REGION Network 98: MENSAJES - AUSENCIA
   RUNG wire#powerrail
      Contact( #Mx_ET151 )
      Contact( #Mx_ET51 )
      wire#w1
      I_Contact( #pHsMx_1 )
      I_Contact( #pHsMx_2 )
      I_Contact( #pHsMx_3 )
      I_Contact( #pHsMx_4 )
      S_SR(operand := #STAT_EnvMens_AMx, r1 := wire#w2)
      Coil( #P_EnvMens_AMx )
   END_RUNG
   RUNG wire#powerrail
      Contact( #Mx_ET161 )
      Contact( #Mx_ET61 )
   END_RUNG wire#w1
   RUNG wire#powerrail
      I_Contact( #Mx_ET151 )
      I_Contact( #Mx_ET161 )
   END_RUNG wire#w2
   // the same network as SCL:
   IF ((#Mx_ET151 AND #Mx_ET51) OR (#Mx_ET161 AND #Mx_ET61)) AND NOT #pHsMx_1 AND NOT #pHsMx_2 AND NOT #pHsMx_3 AND NOT #pHsMx_4 THEN
       #STAT_EnvMens_AMx := TRUE;   // SR flip-flop
   END_IF;
   IF NOT #Mx_ET151 AND NOT #Mx_ET161 THEN #STAT_EnvMens_AMx := FALSE; END_IF;
   #P_EnvMens_AMx := #STAT_EnvMens_AMx;
END_REGION

REGION Network 99: MENSAJES - RECIBIDA LA ORDEN
   RUNG wire#powerrail
      Contact( #Mx_ET150 )
      I_Contact( #Mx_ET50 )
      wire#w1
      Coil( #P_RecepOK_Mx )
   END_RUNG
   RUNG wire#powerrail
      Contact( #Mx_ET160 )
      I_Contact( #Mx_ET60 )
   END_RUNG wire#w1
   // the same network as SCL:
   #P_RecepOK_Mx := (#Mx_ET150 AND NOT #Mx_ET50) OR (#Mx_ET160 AND NOT #Mx_ET60);
END_REGION

REGION Network 100: SALIDAS - Interlock FSS >> PickUp por S1
   RUNG wire#powerrail
      Contact( #Mx_ET60 )
      wire#w1
      Contact( #Pos_TROK )
      Contact( #Pos_TPOK )
      I_Contact( #Activado_Pasarela )
      Contact( #EstadoZona.Marcha_CBx )
      I_Contact( #EstadoVI.Error_Mx )
      I_Contact( #Error_Tx )
      Coil( #MA_PickUpOK_S1 )
   END_RUNG
   RUNG wire#powerrail
      Contact( #Mx_ET61 )
   END_RUNG wire#w1
   RUNG wire#powerrail
      Contact( #Mx_ET261 )
      I_Contact( #EstadoZona.ParoBlando_CBx )
   END_RUNG wire#w1
   // the same network as SCL:
   #MA_PickUpOK_S1 := (#Mx_ET60 OR #Mx_ET61 OR (#Mx_ET261 AND NOT #EstadoZona.ParoBlando_CBx)) AND #Pos_TROK AND #Pos_TPOK AND NOT #Activado_Pasarela AND #EstadoZona.Marcha_CBx AND NOT #EstadoVI.Error_Mx AND NOT #Error_Tx;
END_REGION

REGION Network 101: SALIDAS - Interlock FSS >> PickUp por S3
   RUNG wire#powerrail
      Contact( #Mx_ET50 )
      wire#w1
      Contact( #Pos_TROK )
      Contact( #Pos_TPOK )
      I_Contact( #Activado_Pasarela )
      Contact( #EstadoZona.Marcha_CBx )
      I_Contact( #EstadoVI.Error_Mx )
      I_Contact( #Error_Tx )
      Coil( #MA_PickUpOK_S3 )
   END_RUNG
   RUNG wire#powerrail
      Contact( #Mx_ET51 )
   END_RUNG wire#w1
   RUNG wire#powerrail
      Contact( #Mx_ET261 )
      I_Contact( #EstadoZona.ParoBlando_CBx )
   END_RUNG wire#w1
   // the same network as SCL:
   #MA_PickUpOK_S3 := (#Mx_ET50 OR #Mx_ET51 OR (#Mx_ET261 AND NOT #EstadoZona.ParoBlando_CBx)) AND #Pos_TROK AND #Pos_TPOK AND NOT #Activado_Pasarela AND #EstadoZona.Marcha_CBx AND NOT #EstadoVI.Error_Mx AND NOT #Error_Tx;
END_REGION

REGION Network 102: VARIABLES INTERNAS - AVANCE DE CARGA
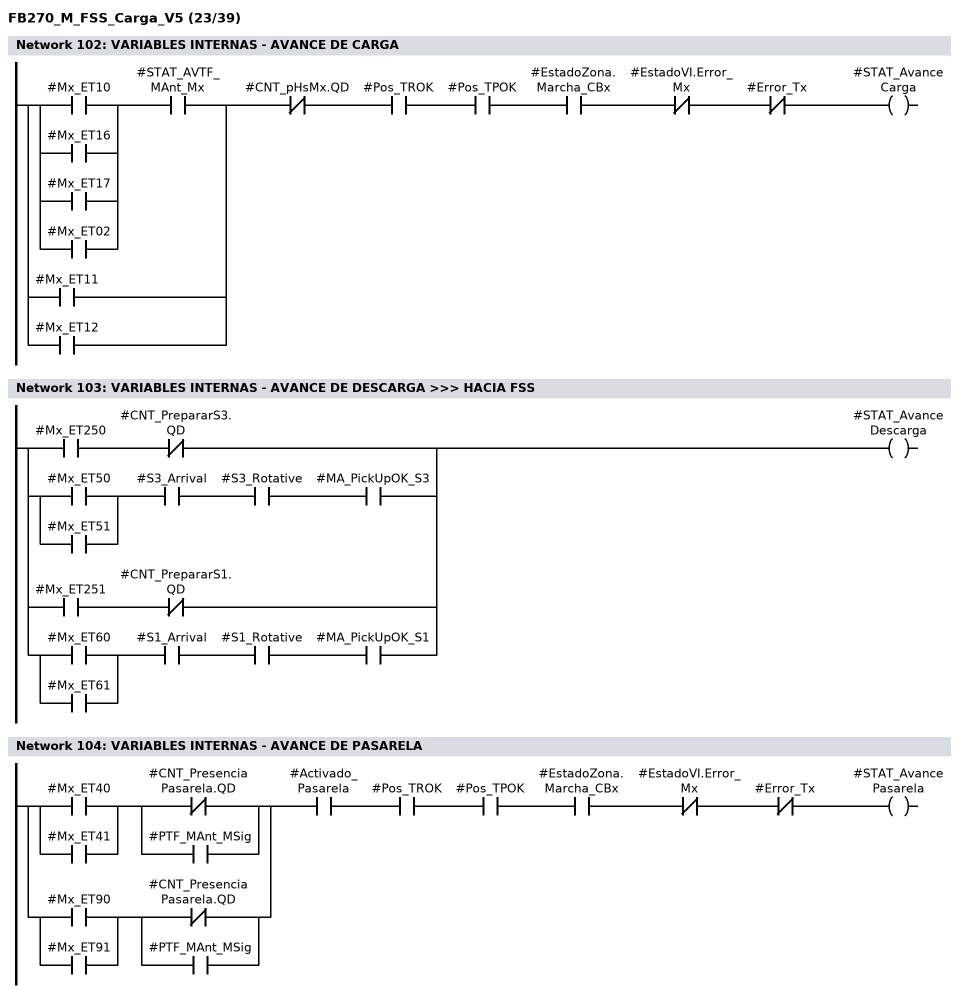
   RUNG wire#powerrail
      Contact( #Mx_ET10 )
      wire#w1
      Contact( #STAT_AVTF_MAnt_Mx )
      wire#w2
      I_Contact( #CNT_pHsMx.QD )
      Contact( #Pos_TROK )
      Contact( #Pos_TPOK )
      Contact( #EstadoZona.Marcha_CBx )
      I_Contact( #EstadoVI.Error_Mx )
      I_Contact( #Error_Tx )
      Coil( #STAT_AvanceCarga )
   END_RUNG
   RUNG wire#powerrail
      Contact( #Mx_ET16 )
   END_RUNG wire#w1
   RUNG wire#powerrail
      Contact( #Mx_ET17 )
   END_RUNG wire#w1
   RUNG wire#powerrail
      Contact( #Mx_ET02 )
   END_RUNG wire#w1
   RUNG wire#powerrail
      Contact( #Mx_ET11 )
   END_RUNG wire#w2
   RUNG wire#powerrail
      Contact( #Mx_ET12 )
   END_RUNG wire#w2
   // the same network as SCL:
   #STAT_AvanceCarga := (((#Mx_ET10 OR #Mx_ET16 OR #Mx_ET17 OR #Mx_ET02) AND #STAT_AVTF_MAnt_Mx) OR #Mx_ET11 OR #Mx_ET12) AND NOT #CNT_pHsMx.QD AND #Pos_TROK AND #Pos_TPOK AND #EstadoZona.Marcha_CBx AND NOT #EstadoVI.Error_Mx AND NOT #Error_Tx;
END_REGION

REGION Network 103: VARIABLES INTERNAS - AVANCE DE DESCARGA >>> HACIA FSS
   RUNG wire#powerrail
      Contact( #Mx_ET250 )
      I_Contact( #CNT_PrepararS3.QD )
      wire#w1
      Coil( #STAT_AvanceDescarga )
   END_RUNG
   RUNG wire#powerrail
      Contact( #Mx_ET50 )
      wire#w2
      Contact( #S3_Arrival )
      Contact( #S3_Rotative )
      Contact( #MA_PickUpOK_S3 )
   END_RUNG wire#w1
   RUNG wire#powerrail
      Contact( #Mx_ET51 )
   END_RUNG wire#w2
   RUNG wire#powerrail
      Contact( #Mx_ET251 )
      I_Contact( #CNT_PrepararS1.QD )
   END_RUNG wire#w1
   RUNG wire#powerrail
      Contact( #Mx_ET60 )
      wire#w3
      Contact( #S1_Arrival )
      Contact( #S1_Rotative )
      Contact( #MA_PickUpOK_S1 )
   END_RUNG wire#w1
   RUNG wire#powerrail
      Contact( #Mx_ET61 )
   END_RUNG wire#w3
   // the same network as SCL:
   #STAT_AvanceDescarga := (#Mx_ET250 AND NOT #CNT_PrepararS3.QD) OR ((#Mx_ET50 OR #Mx_ET51) AND #S3_Arrival AND #S3_Rotative AND #MA_PickUpOK_S3) OR (#Mx_ET251 AND NOT #CNT_PrepararS1.QD) OR ((#Mx_ET60 OR #Mx_ET61) AND #S1_Arrival AND #S1_Rotative AND #MA_PickUpOK_S1);
END_REGION

REGION Network 104: VARIABLES INTERNAS - AVANCE DE PASARELA
   RUNG wire#powerrail
      Contact( #Mx_ET40 )
      wire#w1
      I_Contact( #CNT_PresenciaPasarela.QD )
      wire#w2
      Contact( #Activado_Pasarela )
      Contact( #Pos_TROK )
      Contact( #Pos_TPOK )
      Contact( #EstadoZona.Marcha_CBx )
      I_Contact( #EstadoVI.Error_Mx )
      I_Contact( #Error_Tx )
      Coil( #STAT_AvancePasarela )
   END_RUNG
   RUNG wire#powerrail
      Contact( #Mx_ET41 )
   END_RUNG wire#w1
   RUNG wire#w1
      Contact( #PTF_MAnt_MSig )
   END_RUNG wire#w2
   RUNG wire#powerrail
      Contact( #Mx_ET90 )
      wire#w3
      I_Contact( #CNT_PresenciaPasarela.QD )
   END_RUNG wire#w2
   RUNG wire#powerrail
      Contact( #Mx_ET91 )
   END_RUNG wire#w3
   RUNG wire#w3
      Contact( #PTF_MAnt_MSig )
   END_RUNG wire#w2
   // the same network as SCL:
   #STAT_AvancePasarela := (((#Mx_ET40 OR #Mx_ET41) AND (NOT #CNT_PresenciaPasarela.QD OR #PTF_MAnt_MSig)) OR ((#Mx_ET90 OR #Mx_ET91) AND (NOT #CNT_PresenciaPasarela.QD OR #PTF_MAnt_MSig))) AND #Activado_Pasarela AND #Pos_TROK AND #Pos_TPOK AND #EstadoZona.Marcha_CBx AND NOT #EstadoVI.Error_Mx AND NOT #Error_Tx;
END_REGION

REGION Network 105: VARIABLES INTERNAS - VELOCIDAD BIT 00 >> RODILLOS 00-LenSima 01-Repos 10-Len 11-Rap
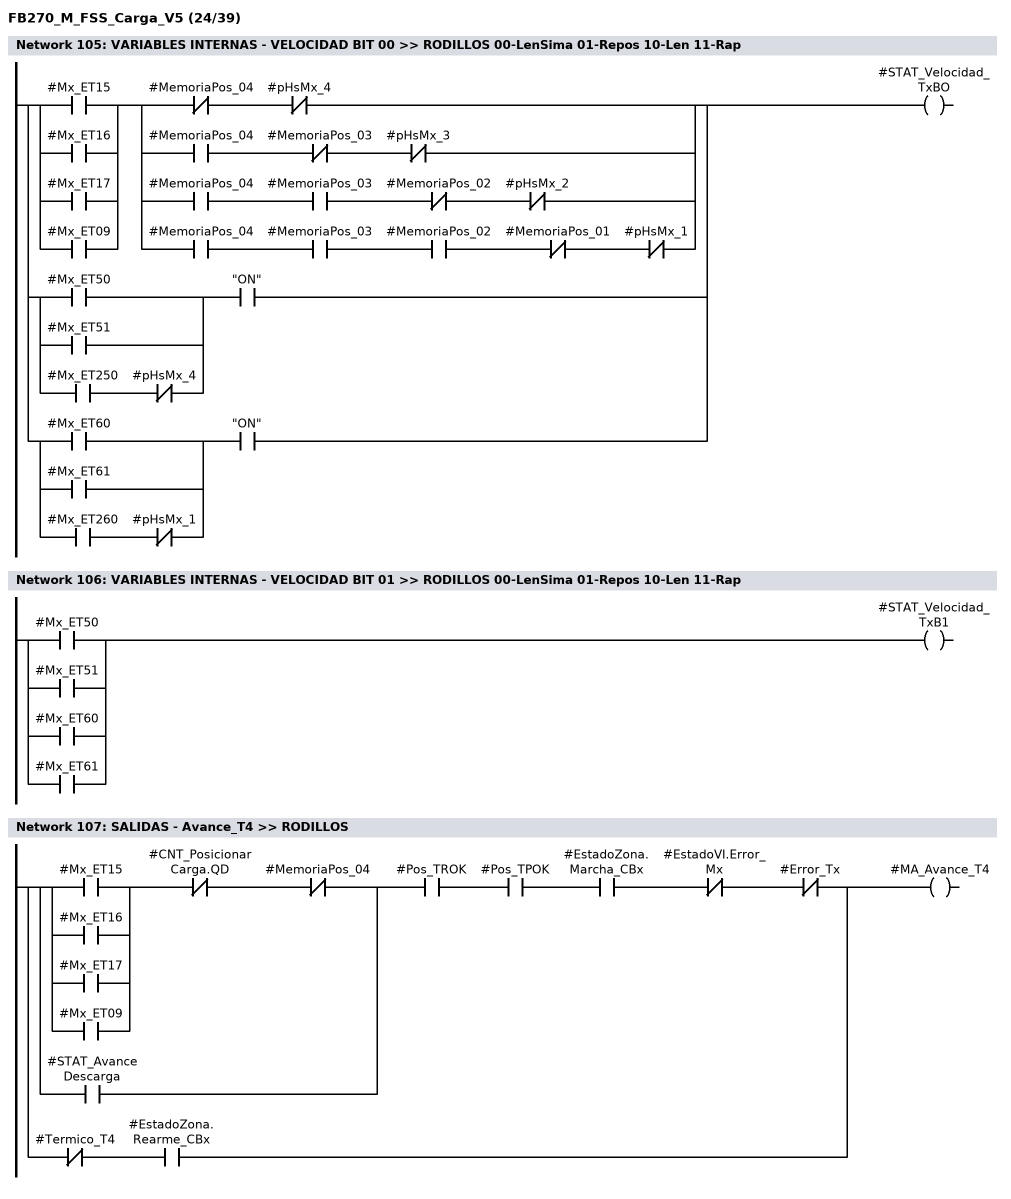
   RUNG wire#powerrail
      Contact( #Mx_ET15 )
      wire#w1
      I_Contact( #MemoriaPos_04 )
      I_Contact( #pHsMx_4 )
      wire#w2
      Coil( #STAT_Velocidad_TxBO )
   END_RUNG
   RUNG wire#powerrail
      Contact( #Mx_ET16 )
   END_RUNG wire#w1
   RUNG wire#powerrail
      Contact( #Mx_ET17 )
   END_RUNG wire#w1
   RUNG wire#powerrail
      Contact( #Mx_ET09 )
   END_RUNG wire#w1
   RUNG wire#w1
      Contact( #MemoriaPos_04 )
      I_Contact( #MemoriaPos_03 )
      I_Contact( #pHsMx_3 )
   END_RUNG wire#w2
   RUNG wire#w1
      Contact( #MemoriaPos_04 )
      Contact( #MemoriaPos_03 )
      I_Contact( #MemoriaPos_02 )
      I_Contact( #pHsMx_2 )
   END_RUNG wire#w2
   RUNG wire#w1
      Contact( #MemoriaPos_04 )
      Contact( #MemoriaPos_03 )
      Contact( #MemoriaPos_02 )
      I_Contact( #MemoriaPos_01 )
      I_Contact( #pHsMx_1 )
   END_RUNG wire#w2
   RUNG wire#powerrail
      Contact( #Mx_ET50 )
      wire#w3
      Contact( "ON" )
   END_RUNG wire#w2
   RUNG wire#powerrail
      Contact( #Mx_ET51 )
   END_RUNG wire#w3
   RUNG wire#powerrail
      Contact( #Mx_ET250 )
      I_Contact( #pHsMx_4 )
   END_RUNG wire#w3
   RUNG wire#powerrail
      Contact( #Mx_ET60 )
      wire#w4
      Contact( "ON" )
   END_RUNG wire#w2
   RUNG wire#powerrail
      Contact( #Mx_ET61 )
   END_RUNG wire#w4
   RUNG wire#powerrail
      Contact( #Mx_ET260 )
      I_Contact( #pHsMx_1 )
   END_RUNG wire#w4
   // the same network as SCL:
   #STAT_Velocidad_TxBO := ((#Mx_ET15 OR #Mx_ET16 OR #Mx_ET17 OR #Mx_ET09) AND ((NOT #MemoriaPos_04 AND NOT #pHsMx_4) OR (#MemoriaPos_04 AND NOT #MemoriaPos_03 AND NOT #pHsMx_3) OR (#MemoriaPos_04 AND #MemoriaPos_03 AND NOT #MemoriaPos_02 AND NOT #pHsMx_2) OR (#MemoriaPos_04 AND #MemoriaPos_03 AND #MemoriaPos_02 AND NOT #MemoriaPos_01 AND NOT #pHsMx_1))) OR ((#Mx_ET50 OR #Mx_ET51 OR (#Mx_ET250 AND NOT #pHsMx_4)) AND "ON") OR ((#Mx_ET60 OR #Mx_ET61 OR (#Mx_ET260 AND NOT #pHsMx_1)) AND "ON");
END_REGION

REGION Network 106: VARIABLES INTERNAS - VELOCIDAD BIT 01 >> RODILLOS 00-LenSima 01-Repos 10-Len 11-Rap
   RUNG wire#powerrail
      Contact( #Mx_ET50 )
      wire#w1
      Coil( #STAT_Velocidad_TxB1 )
   END_RUNG
   RUNG wire#powerrail
      Contact( #Mx_ET51 )
   END_RUNG wire#w1
   RUNG wire#powerrail
      Contact( #Mx_ET60 )
   END_RUNG wire#w1
   RUNG wire#powerrail
      Contact( #Mx_ET61 )
   END_RUNG wire#w1
   // the same network as SCL:
   #STAT_Velocidad_TxB1 := #Mx_ET50 OR #Mx_ET51 OR #Mx_ET60 OR #Mx_ET61;
END_REGION

REGION Network 107: SALIDAS - Avance_T4 >> RODILLOS
   RUNG wire#powerrail
      Contact( #Mx_ET15 )
      wire#w1
      I_Contact( #CNT_PosicionarCarga.QD )
      I_Contact( #MemoriaPos_04 )
      wire#w2
      Contact( #Pos_TROK )
      Contact( #Pos_TPOK )
      Contact( #EstadoZona.Marcha_CBx )
      I_Contact( #EstadoVI.Error_Mx )
      I_Contact( #Error_Tx )
      wire#w3
      Coil( #MA_Avance_T4 )
   END_RUNG
   RUNG wire#powerrail
      Contact( #Mx_ET16 )
   END_RUNG wire#w1
   RUNG wire#powerrail
      Contact( #Mx_ET17 )
   END_RUNG wire#w1
   RUNG wire#powerrail
      Contact( #Mx_ET09 )
   END_RUNG wire#w1
   RUNG wire#powerrail
      Contact( #STAT_AvanceDescarga )
   END_RUNG wire#w2
   RUNG wire#powerrail
      I_Contact( #Termico_T4 )
      Contact( #EstadoZona.Rearme_CBx )
   END_RUNG wire#w3
   // the same network as SCL:
   #MA_Avance_T4 := ((((#Mx_ET15 OR #Mx_ET16 OR #Mx_ET17 OR #Mx_ET09) AND NOT #CNT_PosicionarCarga.QD AND NOT #MemoriaPos_04) OR #STAT_AvanceDescarga) AND #Pos_TROK AND #Pos_TPOK AND #EstadoZona.Marcha_CBx AND NOT #EstadoVI.Error_Mx AND NOT #Error_Tx) OR (NOT #Termico_T4 AND #EstadoZona.Rearme_CBx);
END_REGION

REGION Network 108: SALIDAS - Avance_T3 >> RODILLOS
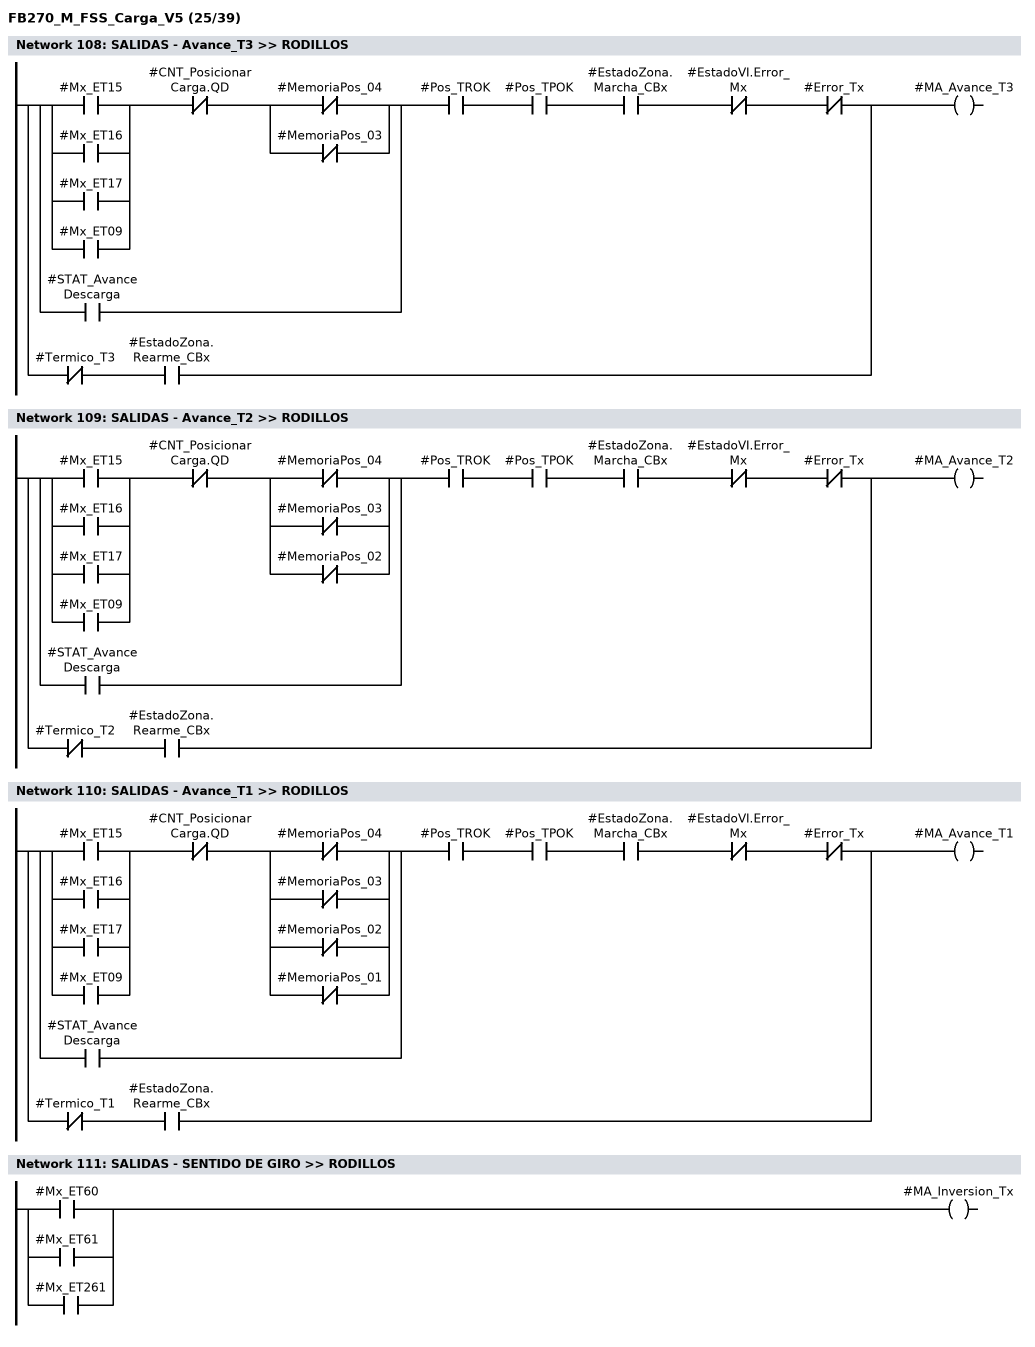
   RUNG wire#powerrail
      Contact( #Mx_ET15 )
      wire#w1
      I_Contact( #CNT_PosicionarCarga.QD )
      wire#w2
      I_Contact( #MemoriaPos_04 )
      wire#w3
      Contact( #Pos_TROK )
      Contact( #Pos_TPOK )
      Contact( #EstadoZona.Marcha_CBx )
      I_Contact( #EstadoVI.Error_Mx )
      I_Contact( #Error_Tx )
      wire#w4
      Coil( #MA_Avance_T3 )
   END_RUNG
   RUNG wire#powerrail
      Contact( #Mx_ET16 )
   END_RUNG wire#w1
   RUNG wire#powerrail
      Contact( #Mx_ET17 )
   END_RUNG wire#w1
   RUNG wire#powerrail
      Contact( #Mx_ET09 )
   END_RUNG wire#w1
   RUNG wire#w2
      I_Contact( #MemoriaPos_03 )
   END_RUNG wire#w3
   RUNG wire#powerrail
      Contact( #STAT_AvanceDescarga )
   END_RUNG wire#w3
   RUNG wire#powerrail
      I_Contact( #Termico_T3 )
      Contact( #EstadoZona.Rearme_CBx )
   END_RUNG wire#w4
   // the same network as SCL:
   #MA_Avance_T3 := ((((#Mx_ET15 OR #Mx_ET16 OR #Mx_ET17 OR #Mx_ET09) AND NOT #CNT_PosicionarCarga.QD AND (NOT #MemoriaPos_04 OR NOT #MemoriaPos_03)) OR #STAT_AvanceDescarga) AND #Pos_TROK AND #Pos_TPOK AND #EstadoZona.Marcha_CBx AND NOT #EstadoVI.Error_Mx AND NOT #Error_Tx) OR (NOT #Termico_T3 AND #EstadoZona.Rearme_CBx);
END_REGION

REGION Network 109: SALIDAS - Avance_T2 >> RODILLOS
   RUNG wire#powerrail
      Contact( #Mx_ET15 )
      wire#w1
      I_Contact( #CNT_PosicionarCarga.QD )
      wire#w2
      I_Contact( #MemoriaPos_04 )
      wire#w3
      Contact( #Pos_TROK )
      Contact( #Pos_TPOK )
      Contact( #EstadoZona.Marcha_CBx )
      I_Contact( #EstadoVI.Error_Mx )
      I_Contact( #Error_Tx )
      wire#w4
      Coil( #MA_Avance_T2 )
   END_RUNG
   RUNG wire#powerrail
      Contact( #Mx_ET16 )
   END_RUNG wire#w1
   RUNG wire#powerrail
      Contact( #Mx_ET17 )
   END_RUNG wire#w1
   RUNG wire#powerrail
      Contact( #Mx_ET09 )
   END_RUNG wire#w1
   RUNG wire#w2
      I_Contact( #MemoriaPos_03 )
   END_RUNG wire#w3
   RUNG wire#w2
      I_Contact( #MemoriaPos_02 )
   END_RUNG wire#w3
   RUNG wire#powerrail
      Contact( #STAT_AvanceDescarga )
   END_RUNG wire#w3
   RUNG wire#powerrail
      I_Contact( #Termico_T2 )
      Contact( #EstadoZona.Rearme_CBx )
   END_RUNG wire#w4
   // the same network as SCL:
   #MA_Avance_T2 := ((((#Mx_ET15 OR #Mx_ET16 OR #Mx_ET17 OR #Mx_ET09) AND NOT #CNT_PosicionarCarga.QD AND (NOT #MemoriaPos_04 OR NOT #MemoriaPos_03 OR NOT #MemoriaPos_02)) OR #STAT_AvanceDescarga) AND #Pos_TROK AND #Pos_TPOK AND #EstadoZona.Marcha_CBx AND NOT #EstadoVI.Error_Mx AND NOT #Error_Tx) OR (NOT #Termico_T2 AND #EstadoZona.Rearme_CBx);
END_REGION

REGION Network 110: SALIDAS - Avance_T1 >> RODILLOS
   RUNG wire#powerrail
      Contact( #Mx_ET15 )
      wire#w1
      I_Contact( #CNT_PosicionarCarga.QD )
      wire#w2
      I_Contact( #MemoriaPos_04 )
      wire#w3
      Contact( #Pos_TROK )
      Contact( #Pos_TPOK )
      Contact( #EstadoZona.Marcha_CBx )
      I_Contact( #EstadoVI.Error_Mx )
      I_Contact( #Error_Tx )
      wire#w4
      Coil( #MA_Avance_T1 )
   END_RUNG
   RUNG wire#powerrail
      Contact( #Mx_ET16 )
   END_RUNG wire#w1
   RUNG wire#powerrail
      Contact( #Mx_ET17 )
   END_RUNG wire#w1
   RUNG wire#powerrail
      Contact( #Mx_ET09 )
   END_RUNG wire#w1
   RUNG wire#w2
      I_Contact( #MemoriaPos_03 )
   END_RUNG wire#w3
   RUNG wire#w2
      I_Contact( #MemoriaPos_02 )
   END_RUNG wire#w3
   RUNG wire#w2
      I_Contact( #MemoriaPos_01 )
   END_RUNG wire#w3
   RUNG wire#powerrail
      Contact( #STAT_AvanceDescarga )
   END_RUNG wire#w3
   RUNG wire#powerrail
      I_Contact( #Termico_T1 )
      Contact( #EstadoZona.Rearme_CBx )
   END_RUNG wire#w4
   // the same network as SCL:
   #MA_Avance_T1 := ((((#Mx_ET15 OR #Mx_ET16 OR #Mx_ET17 OR #Mx_ET09) AND NOT #CNT_PosicionarCarga.QD AND (NOT #MemoriaPos_04 OR NOT #MemoriaPos_03 OR NOT #MemoriaPos_02 OR NOT #MemoriaPos_01)) OR #STAT_AvanceDescarga) AND #Pos_TROK AND #Pos_TPOK AND #EstadoZona.Marcha_CBx AND NOT #EstadoVI.Error_Mx AND NOT #Error_Tx) OR (NOT #Termico_T1 AND #EstadoZona.Rearme_CBx);
END_REGION

REGION Network 111: SALIDAS - SENTIDO DE GIRO >> RODILLOS
   RUNG wire#powerrail
      Contact( #Mx_ET60 )
      wire#w1
      Coil( #MA_Inversion_Tx )
   END_RUNG
   RUNG wire#powerrail
      Contact( #Mx_ET61 )
   END_RUNG wire#w1
   RUNG wire#powerrail
      Contact( #Mx_ET261 )
   END_RUNG wire#w1
   // the same network as SCL:
   #MA_Inversion_Tx := #Mx_ET60 OR #Mx_ET61 OR #Mx_ET261;
END_REGION

REGION Network 112: SALIDAS - VELOCIDAD ANALOGICA >> RODILLOS
   // 25T229A_03 
   // Plantilla_Avance_E1S3_SinVariador_1Mesas.
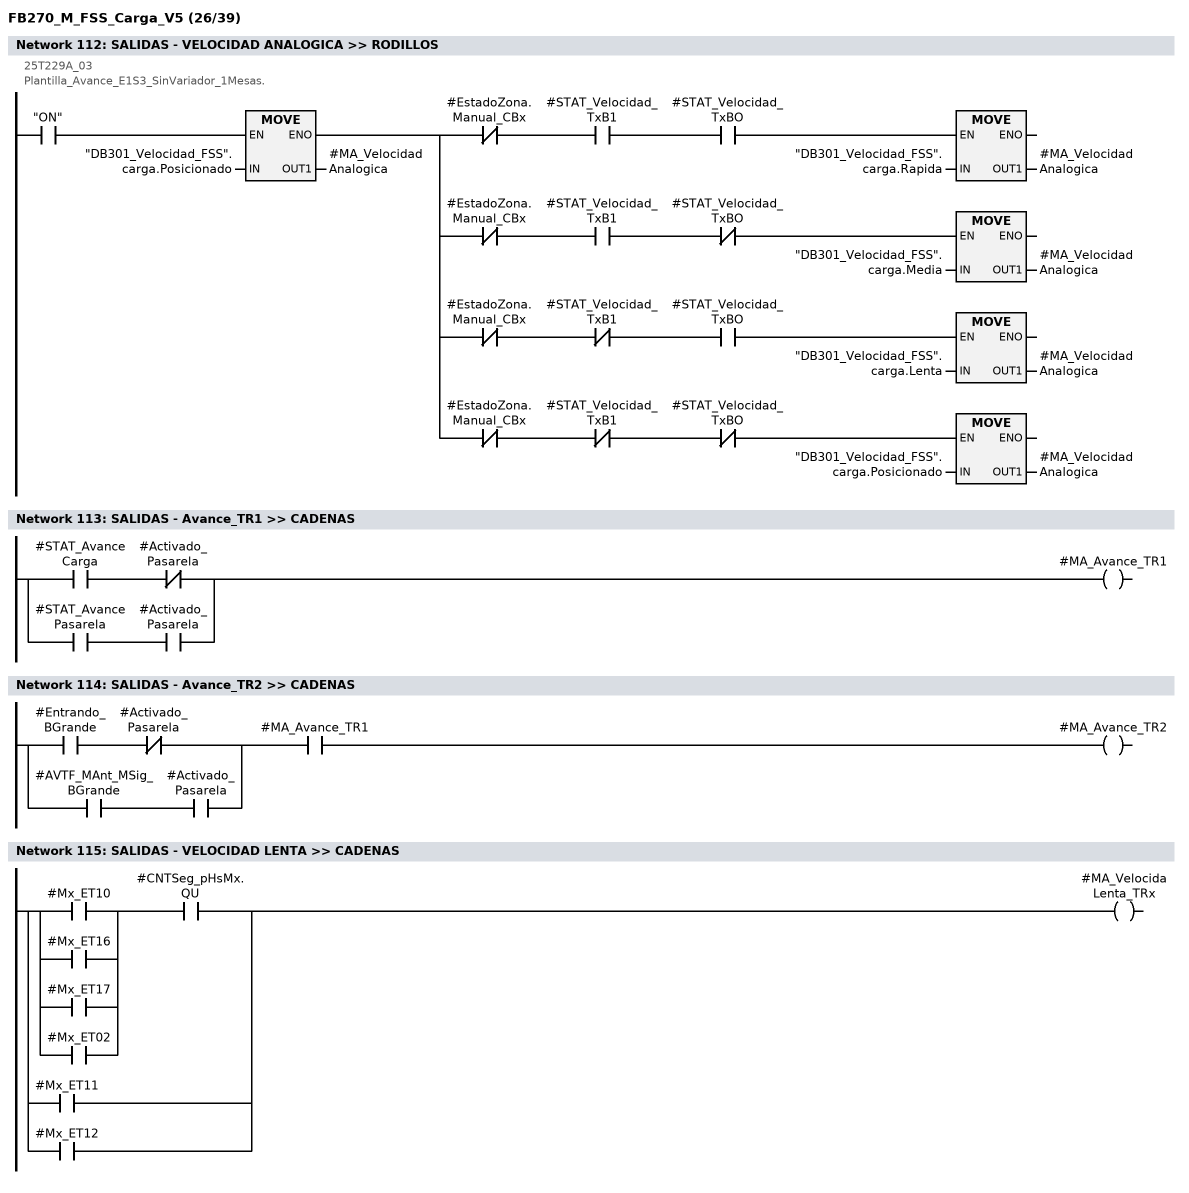
   RUNG wire#powerrail
      Contact( "ON" )
      { S7_GenerateENO := "TRUE" } Move(in := "DB301_Velocidad_FSS".carga.Posicionado, out1 => #MA_VelocidadAnalogica)
      wire#w1
      I_Contact( #EstadoZona.Manual_CBx )
      Contact( #STAT_Velocidad_TxB1 )
      Contact( #STAT_Velocidad_TxBO )
      { S7_GenerateENO := "TRUE" } Move(in := "DB301_Velocidad_FSS".carga.Rapida, out1 => #MA_VelocidadAnalogica)
   END_RUNG
   RUNG wire#w1
      I_Contact( #EstadoZona.Manual_CBx )
      Contact( #STAT_Velocidad_TxB1 )
      I_Contact( #STAT_Velocidad_TxBO )
      { S7_GenerateENO := "TRUE" } Move(in := "DB301_Velocidad_FSS".carga.Media, out1 => #MA_VelocidadAnalogica)
   END_RUNG
   RUNG wire#w1
      I_Contact( #EstadoZona.Manual_CBx )
      I_Contact( #STAT_Velocidad_TxB1 )
      Contact( #STAT_Velocidad_TxBO )
      { S7_GenerateENO := "TRUE" } Move(in := "DB301_Velocidad_FSS".carga.Lenta, out1 => #MA_VelocidadAnalogica)
   END_RUNG
   RUNG wire#w1
      I_Contact( #EstadoZona.Manual_CBx )
      I_Contact( #STAT_Velocidad_TxB1 )
      I_Contact( #STAT_Velocidad_TxBO )
      { S7_GenerateENO := "TRUE" } Move(in := "DB301_Velocidad_FSS".carga.Posicionado, out1 => #MA_VelocidadAnalogica)
   END_RUNG
   // the same network as SCL:
   // ENO of a box is taken as its EN; it also drops when the box reports an error
   IF "ON" THEN #MA_VelocidadAnalogica := "DB301_Velocidad_FSS".carga.Posicionado; END_IF;
   IF "ON" AND NOT #EstadoZona.Manual_CBx AND #STAT_Velocidad_TxB1 AND #STAT_Velocidad_TxBO THEN
       #MA_VelocidadAnalogica := "DB301_Velocidad_FSS".carga.Rapida;
   END_IF;
   IF "ON" AND NOT #EstadoZona.Manual_CBx AND #STAT_Velocidad_TxB1 AND NOT #STAT_Velocidad_TxBO THEN
       #MA_VelocidadAnalogica := "DB301_Velocidad_FSS".carga.Media;
   END_IF;
   IF "ON" AND NOT #EstadoZona.Manual_CBx AND NOT #STAT_Velocidad_TxB1 AND #STAT_Velocidad_TxBO THEN
       #MA_VelocidadAnalogica := "DB301_Velocidad_FSS".carga.Lenta;
   END_IF;
   IF "ON" AND NOT #EstadoZona.Manual_CBx AND NOT #STAT_Velocidad_TxB1 AND NOT #STAT_Velocidad_TxBO THEN
       #MA_VelocidadAnalogica := "DB301_Velocidad_FSS".carga.Posicionado;
   END_IF;
END_REGION

REGION Network 113: SALIDAS - Avance_TR1 >> CADENAS
   RUNG wire#powerrail
      Contact( #STAT_AvanceCarga )
      I_Contact( #Activado_Pasarela )
      wire#w1
      Coil( #MA_Avance_TR1 )
   END_RUNG
   RUNG wire#powerrail
      Contact( #STAT_AvancePasarela )
      Contact( #Activado_Pasarela )
   END_RUNG wire#w1
   // the same network as SCL:
   #MA_Avance_TR1 := (#STAT_AvanceCarga AND NOT #Activado_Pasarela) OR (#STAT_AvancePasarela AND #Activado_Pasarela);
END_REGION

REGION Network 114: SALIDAS - Avance_TR2 >> CADENAS
   RUNG wire#powerrail
      Contact( #Entrando_BGrande )
      I_Contact( #Activado_Pasarela )
      wire#w1
      Contact( #MA_Avance_TR1 )
      Coil( #MA_Avance_TR2 )
   END_RUNG
   RUNG wire#powerrail
      Contact( #AVTF_MAnt_MSig_BGrande )
      Contact( #Activado_Pasarela )
   END_RUNG wire#w1
   // the same network as SCL:
   #MA_Avance_TR2 := ((#Entrando_BGrande AND NOT #Activado_Pasarela) OR (#AVTF_MAnt_MSig_BGrande AND #Activado_Pasarela)) AND #MA_Avance_TR1;
END_REGION

REGION Network 115: SALIDAS - VELOCIDAD LENTA >> CADENAS
   RUNG wire#powerrail
      Contact( #Mx_ET10 )
      wire#w1
      Contact( #CNTSeg_pHsMx.QU )
      wire#w2
      Coil( #MA_VelocidaLenta_TRx )
   END_RUNG
   RUNG wire#powerrail
      Contact( #Mx_ET16 )
   END_RUNG wire#w1
   RUNG wire#powerrail
      Contact( #Mx_ET17 )
   END_RUNG wire#w1
   RUNG wire#powerrail
      Contact( #Mx_ET02 )
   END_RUNG wire#w1
   RUNG wire#powerrail
      Contact( #Mx_ET11 )
   END_RUNG wire#w2
   RUNG wire#powerrail
      Contact( #Mx_ET12 )
   END_RUNG wire#w2
   // the same network as SCL:
   #MA_VelocidaLenta_TRx := ((#Mx_ET10 OR #Mx_ET16 OR #Mx_ET17 OR #Mx_ET02) AND #CNTSeg_pHsMx.QU) OR #Mx_ET11 OR #Mx_ET12;
END_REGION

REGION Network 116: SALIDAS - SUBIR TRANSTER TR1 (Neumatica)
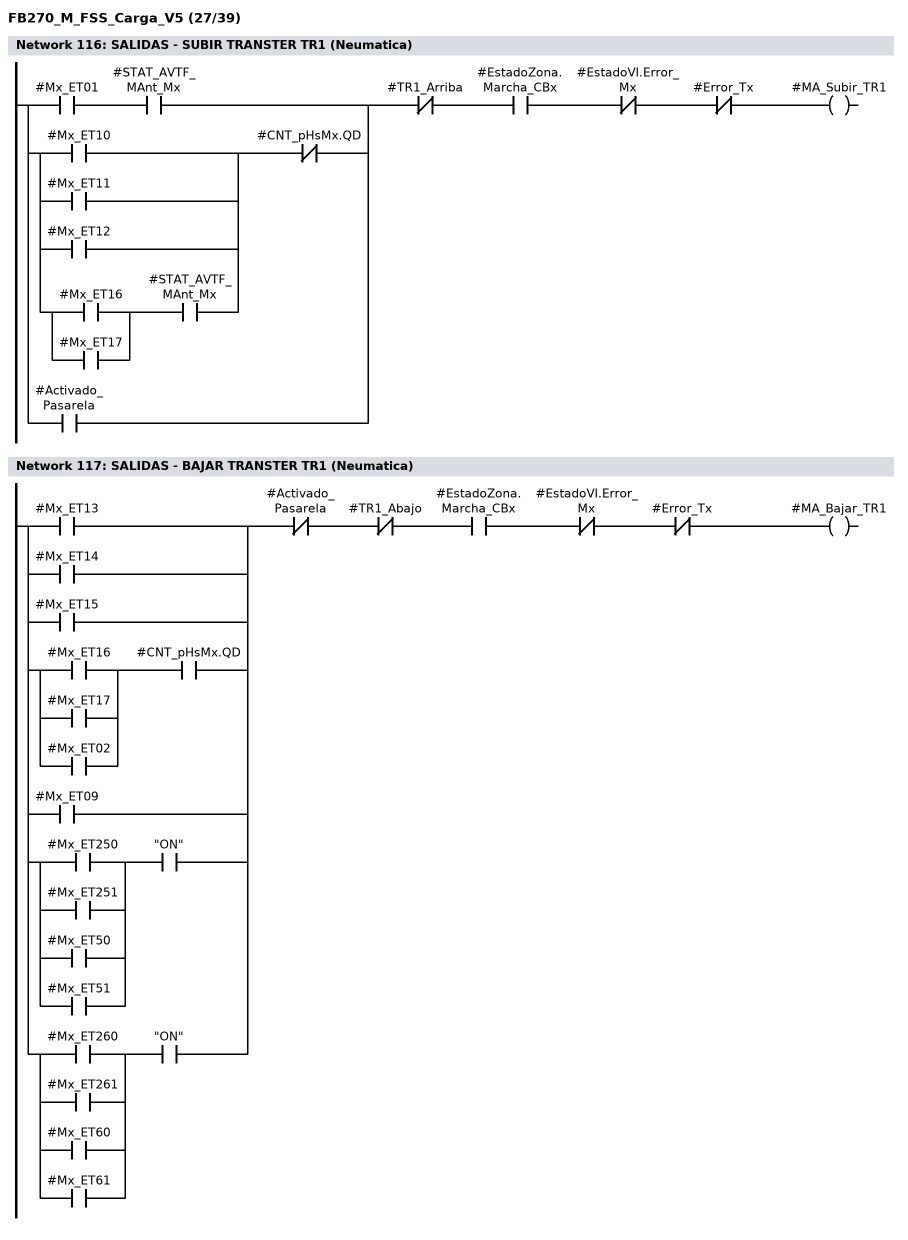
   RUNG wire#powerrail
      Contact( #Mx_ET01 )
      Contact( #STAT_AVTF_MAnt_Mx )
      wire#w1
      I_Contact( #TR1_Arriba )
      Contact( #EstadoZona.Marcha_CBx )
      I_Contact( #EstadoVI.Error_Mx )
      I_Contact( #Error_Tx )
      Coil( #MA_Subir_TR1 )
   END_RUNG
   RUNG wire#powerrail
      Contact( #Mx_ET10 )
      wire#w2
      I_Contact( #CNT_pHsMx.QD )
   END_RUNG wire#w1
   RUNG wire#powerrail
      Contact( #Mx_ET11 )
   END_RUNG wire#w2
   RUNG wire#powerrail
      Contact( #Mx_ET12 )
   END_RUNG wire#w2
   RUNG wire#powerrail
      Contact( #Mx_ET16 )
      wire#w3
      Contact( #STAT_AVTF_MAnt_Mx )
   END_RUNG wire#w2
   RUNG wire#powerrail
      Contact( #Mx_ET17 )
   END_RUNG wire#w3
   RUNG wire#powerrail
      Contact( #Activado_Pasarela )
   END_RUNG wire#w1
   // the same network as SCL:
   #MA_Subir_TR1 := ((#Mx_ET01 AND #STAT_AVTF_MAnt_Mx) OR ((#Mx_ET10 OR #Mx_ET11 OR #Mx_ET12 OR ((#Mx_ET16 OR #Mx_ET17) AND #STAT_AVTF_MAnt_Mx)) AND NOT #CNT_pHsMx.QD) OR #Activado_Pasarela) AND NOT #TR1_Arriba AND #EstadoZona.Marcha_CBx AND NOT #EstadoVI.Error_Mx AND NOT #Error_Tx;
END_REGION

REGION Network 117: SALIDAS - BAJAR TRANSTER TR1 (Neumatica)
   RUNG wire#powerrail
      Contact( #Mx_ET13 )
      wire#w1
      I_Contact( #Activado_Pasarela )
      I_Contact( #TR1_Abajo )
      Contact( #EstadoZona.Marcha_CBx )
      I_Contact( #EstadoVI.Error_Mx )
      I_Contact( #Error_Tx )
      Coil( #MA_Bajar_TR1 )
   END_RUNG
   RUNG wire#powerrail
      Contact( #Mx_ET14 )
   END_RUNG wire#w1
   RUNG wire#powerrail
      Contact( #Mx_ET15 )
   END_RUNG wire#w1
   RUNG wire#powerrail
      Contact( #Mx_ET16 )
      wire#w2
      Contact( #CNT_pHsMx.QD )
   END_RUNG wire#w1
   RUNG wire#powerrail
      Contact( #Mx_ET17 )
   END_RUNG wire#w2
   RUNG wire#powerrail
      Contact( #Mx_ET02 )
   END_RUNG wire#w2
   RUNG wire#powerrail
      Contact( #Mx_ET09 )
   END_RUNG wire#w1
   RUNG wire#powerrail
      Contact( #Mx_ET250 )
      wire#w3
      Contact( "ON" )
   END_RUNG wire#w1
   RUNG wire#powerrail
      Contact( #Mx_ET251 )
   END_RUNG wire#w3
   RUNG wire#powerrail
      Contact( #Mx_ET50 )
   END_RUNG wire#w3
   RUNG wire#powerrail
      Contact( #Mx_ET51 )
   END_RUNG wire#w3
   RUNG wire#powerrail
      Contact( #Mx_ET260 )
      wire#w4
      Contact( "ON" )
   END_RUNG wire#w1
   RUNG wire#powerrail
      Contact( #Mx_ET261 )
   END_RUNG wire#w4
   RUNG wire#powerrail
      Contact( #Mx_ET60 )
   END_RUNG wire#w4
   RUNG wire#powerrail
      Contact( #Mx_ET61 )
   END_RUNG wire#w4
   // the same network as SCL:
   #MA_Bajar_TR1 := (#Mx_ET13 OR #Mx_ET14 OR #Mx_ET15 OR ((#Mx_ET16 OR #Mx_ET17 OR #Mx_ET02) AND #CNT_pHsMx.QD) OR #Mx_ET09 OR ((#Mx_ET250 OR #Mx_ET251 OR #Mx_ET50 OR #Mx_ET51) AND "ON") OR ((#Mx_ET260 OR #Mx_ET261 OR #Mx_ET60 OR #Mx_ET61) AND "ON")) AND NOT #Activado_Pasarela AND NOT #TR1_Abajo AND #EstadoZona.Marcha_CBx AND NOT #EstadoVI.Error_Mx AND NOT #Error_Tx;
END_REGION

REGION Network 118: SALIDAS - SUBIR TRANSTER TR2 (Neumatica)
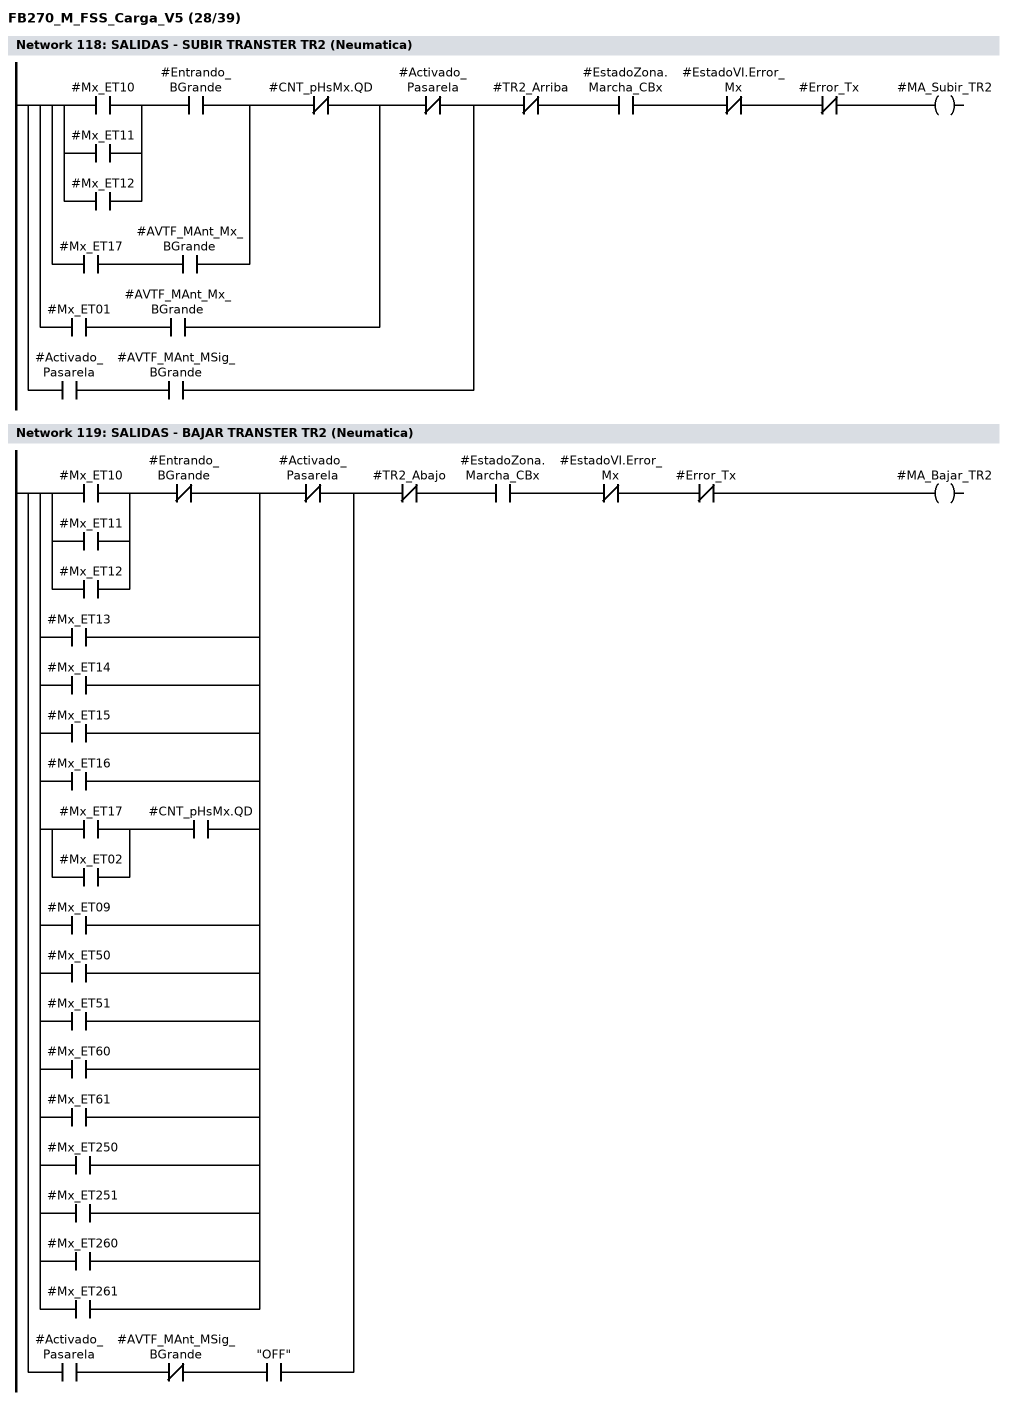
   RUNG wire#powerrail
      Contact( #Mx_ET10 )
      wire#w1
      Contact( #Entrando_BGrande )
      wire#w2
      I_Contact( #CNT_pHsMx.QD )
      wire#w3
      I_Contact( #Activado_Pasarela )
      wire#w4
      I_Contact( #TR2_Arriba )
      Contact( #EstadoZona.Marcha_CBx )
      I_Contact( #EstadoVI.Error_Mx )
      I_Contact( #Error_Tx )
      Coil( #MA_Subir_TR2 )
   END_RUNG
   RUNG wire#powerrail
      Contact( #Mx_ET11 )
   END_RUNG wire#w1
   RUNG wire#powerrail
      Contact( #Mx_ET12 )
   END_RUNG wire#w1
   RUNG wire#powerrail
      Contact( #Mx_ET17 )
      Contact( #AVTF_MAnt_Mx_BGrande )
   END_RUNG wire#w2
   RUNG wire#powerrail
      Contact( #Mx_ET01 )
      Contact( #AVTF_MAnt_Mx_BGrande )
   END_RUNG wire#w3
   RUNG wire#powerrail
      Contact( #Activado_Pasarela )
      Contact( #AVTF_MAnt_MSig_BGrande )
   END_RUNG wire#w4
   // the same network as SCL:
   #MA_Subir_TR2 := (((((((#Mx_ET10 OR #Mx_ET11 OR #Mx_ET12) AND #Entrando_BGrande) OR (#Mx_ET17 AND #AVTF_MAnt_Mx_BGrande)) AND NOT #CNT_pHsMx.QD) OR (#Mx_ET01 AND #AVTF_MAnt_Mx_BGrande)) AND NOT #Activado_Pasarela) OR (#Activado_Pasarela AND #AVTF_MAnt_MSig_BGrande)) AND NOT #TR2_Arriba AND #EstadoZona.Marcha_CBx AND NOT #EstadoVI.Error_Mx AND NOT #Error_Tx;
END_REGION

REGION Network 119: SALIDAS - BAJAR TRANSTER TR2 (Neumatica)
   RUNG wire#powerrail
      Contact( #Mx_ET10 )
      wire#w1
      I_Contact( #Entrando_BGrande )
      wire#w2
      I_Contact( #Activado_Pasarela )
      wire#w4
      I_Contact( #TR2_Abajo )
      Contact( #EstadoZona.Marcha_CBx )
      I_Contact( #EstadoVI.Error_Mx )
      I_Contact( #Error_Tx )
      Coil( #MA_Bajar_TR2 )
   END_RUNG
   RUNG wire#powerrail
      Contact( #Mx_ET11 )
   END_RUNG wire#w1
   RUNG wire#powerrail
      Contact( #Mx_ET12 )
   END_RUNG wire#w1
   RUNG wire#powerrail
      Contact( #Mx_ET13 )
   END_RUNG wire#w2
   RUNG wire#powerrail
      Contact( #Mx_ET14 )
   END_RUNG wire#w2
   RUNG wire#powerrail
      Contact( #Mx_ET15 )
   END_RUNG wire#w2
   RUNG wire#powerrail
      Contact( #Mx_ET16 )
   END_RUNG wire#w2
   RUNG wire#powerrail
      Contact( #Mx_ET17 )
      wire#w3
      Contact( #CNT_pHsMx.QD )
   END_RUNG wire#w2
   RUNG wire#powerrail
      Contact( #Mx_ET02 )
   END_RUNG wire#w3
   RUNG wire#powerrail
      Contact( #Mx_ET09 )
   END_RUNG wire#w2
   RUNG wire#powerrail
      Contact( #Mx_ET50 )
   END_RUNG wire#w2
   RUNG wire#powerrail
      Contact( #Mx_ET51 )
   END_RUNG wire#w2
   RUNG wire#powerrail
      Contact( #Mx_ET60 )
   END_RUNG wire#w2
   RUNG wire#powerrail
      Contact( #Mx_ET61 )
   END_RUNG wire#w2
   RUNG wire#powerrail
      Contact( #Mx_ET250 )
   END_RUNG wire#w2
   RUNG wire#powerrail
      Contact( #Mx_ET251 )
   END_RUNG wire#w2
   RUNG wire#powerrail
      Contact( #Mx_ET260 )
   END_RUNG wire#w2
   RUNG wire#powerrail
      Contact( #Mx_ET261 )
   END_RUNG wire#w2
   RUNG wire#powerrail
      Contact( #Activado_Pasarela )
      I_Contact( #AVTF_MAnt_MSig_BGrande )
      Contact( "OFF" )
   END_RUNG wire#w4
   // the same network as SCL:
   #MA_Bajar_TR2 := (((((#Mx_ET10 OR #Mx_ET11 OR #Mx_ET12) AND NOT #Entrando_BGrande) OR #Mx_ET13 OR #Mx_ET14 OR #Mx_ET15 OR #Mx_ET16 OR ((#Mx_ET17 OR #Mx_ET02) AND #CNT_pHsMx.QD) OR #Mx_ET09 OR #Mx_ET50 OR #Mx_ET51 OR #Mx_ET60 OR #Mx_ET61 OR #Mx_ET250 OR #Mx_ET251 OR #Mx_ET260 OR #Mx_ET261) AND NOT #Activado_Pasarela) OR (#Activado_Pasarela AND NOT #AVTF_MAnt_MSig_BGrande AND "OFF")) AND NOT #TR2_Abajo AND #EstadoZona.Marcha_CBx AND NOT #EstadoVI.Error_Mx AND NOT #Error_Tx;
END_REGION

REGION Network 120: TMP - Espera En Tension
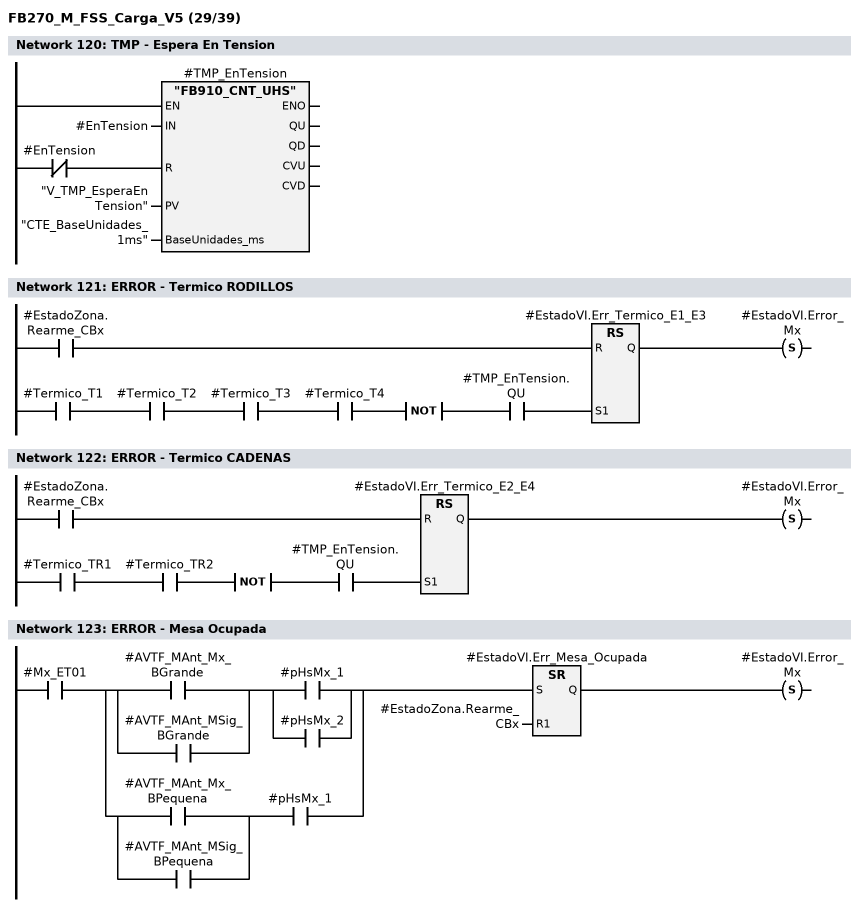
   RUNG wire#powerrail
      #TMP_EnTension(R := wire#w1, IN := #EnTension, PV := "V_TMP_EsperaEnTension", BaseUnidades_ms := "CTE_BaseUnidades_1ms", QU =>, QD =>, CVU =>, CVD =>)
   END_RUNG
   RUNG wire#powerrail
      I_Contact( #EnTension )
   END_RUNG wire#w1
   // the same network as SCL:
   #TMP_EnTension(IN := #EnTension,   // "FB910_CNT_UHS"
                  R := NOT #EnTension,
                  PV := "V_TMP_EsperaEnTension",
                  BaseUnidades_ms := "CTE_BaseUnidades_1ms");
END_REGION

REGION Network 121: ERROR - Termico RODILLOS
   RUNG wire#powerrail
      Contact( #EstadoZona.Rearme_CBx )
      S_RS(operand := #EstadoVI.Err_Termico_E1_E3, s1 := wire#w1)
      S_Coil( #EstadoVI.Error_Mx )
   END_RUNG
   RUNG wire#powerrail
      Contact( #Termico_T1 )
      Contact( #Termico_T2 )
      Contact( #Termico_T3 )
      Contact( #Termico_T4 )
      Not()
      Contact( #TMP_EnTension.QU )
   END_RUNG wire#w1
   // the same network as SCL:
   IF #EstadoZona.Rearme_CBx THEN
       #EstadoVI.Err_Termico_E1_E3 := FALSE;   // RS flip-flop
   END_IF;
   IF NOT (#Termico_T1 AND #Termico_T2 AND #Termico_T3 AND #Termico_T4) AND #TMP_EnTension.QU THEN
       #EstadoVI.Err_Termico_E1_E3 := TRUE;
   END_IF;
   IF #EstadoVI.Err_Termico_E1_E3 THEN #EstadoVI.Error_Mx := TRUE; END_IF;
END_REGION

REGION Network 122: ERROR - Termico CADENAS
   RUNG wire#powerrail
      Contact( #EstadoZona.Rearme_CBx )
      S_RS(operand := #EstadoVI.Err_Termico_E2_E4, s1 := wire#w1)
      S_Coil( #EstadoVI.Error_Mx )
   END_RUNG
   RUNG wire#powerrail
      Contact( #Termico_TR1 )
      Contact( #Termico_TR2 )
      Not()
      Contact( #TMP_EnTension.QU )
   END_RUNG wire#w1
   // the same network as SCL:
   IF #EstadoZona.Rearme_CBx THEN
       #EstadoVI.Err_Termico_E2_E4 := FALSE;   // RS flip-flop
   END_IF;
   IF NOT (#Termico_TR1 AND #Termico_TR2) AND #TMP_EnTension.QU THEN
       #EstadoVI.Err_Termico_E2_E4 := TRUE;
   END_IF;
   IF #EstadoVI.Err_Termico_E2_E4 THEN #EstadoVI.Error_Mx := TRUE; END_IF;
END_REGION

REGION Network 123: ERROR - Mesa Ocupada
   RUNG wire#powerrail
      Contact( #Mx_ET01 )
      wire#w1
      Contact( #AVTF_MAnt_Mx_BGrande )
      wire#w2
      Contact( #pHsMx_1 )
      wire#w3
      S_SR(operand := #EstadoVI.Err_Mesa_Ocupada, r1 := #EstadoZona.Rearme_CBx)
      S_Coil( #EstadoVI.Error_Mx )
   END_RUNG
   RUNG wire#w1
      Contact( #AVTF_MAnt_MSig_BGrande )
   END_RUNG wire#w2
   RUNG wire#w2
      Contact( #pHsMx_2 )
   END_RUNG wire#w3
   RUNG wire#w1
      Contact( #AVTF_MAnt_Mx_BPequena )
      wire#w4
      Contact( #pHsMx_1 )
   END_RUNG wire#w3
   RUNG wire#w1
      Contact( #AVTF_MAnt_MSig_BPequena )
   END_RUNG wire#w4
   // the same network as SCL:
   IF #Mx_ET01 AND (((#AVTF_MAnt_Mx_BGrande OR #AVTF_MAnt_MSig_BGrande) AND (#pHsMx_1 OR #pHsMx_2)) OR ((#AVTF_MAnt_Mx_BPequena OR #AVTF_MAnt_MSig_BPequena) AND #pHsMx_1)) THEN
       #EstadoVI.Err_Mesa_Ocupada := TRUE;   // SR flip-flop
   END_IF;
   IF #EstadoZona.Rearme_CBx THEN #EstadoVI.Err_Mesa_Ocupada := FALSE; END_IF;
   IF #EstadoVI.Err_Mesa_Ocupada THEN #EstadoVI.Error_Mx := TRUE; END_IF;
END_REGION

REGION Network 124: CNT - ERROR - Arrastre
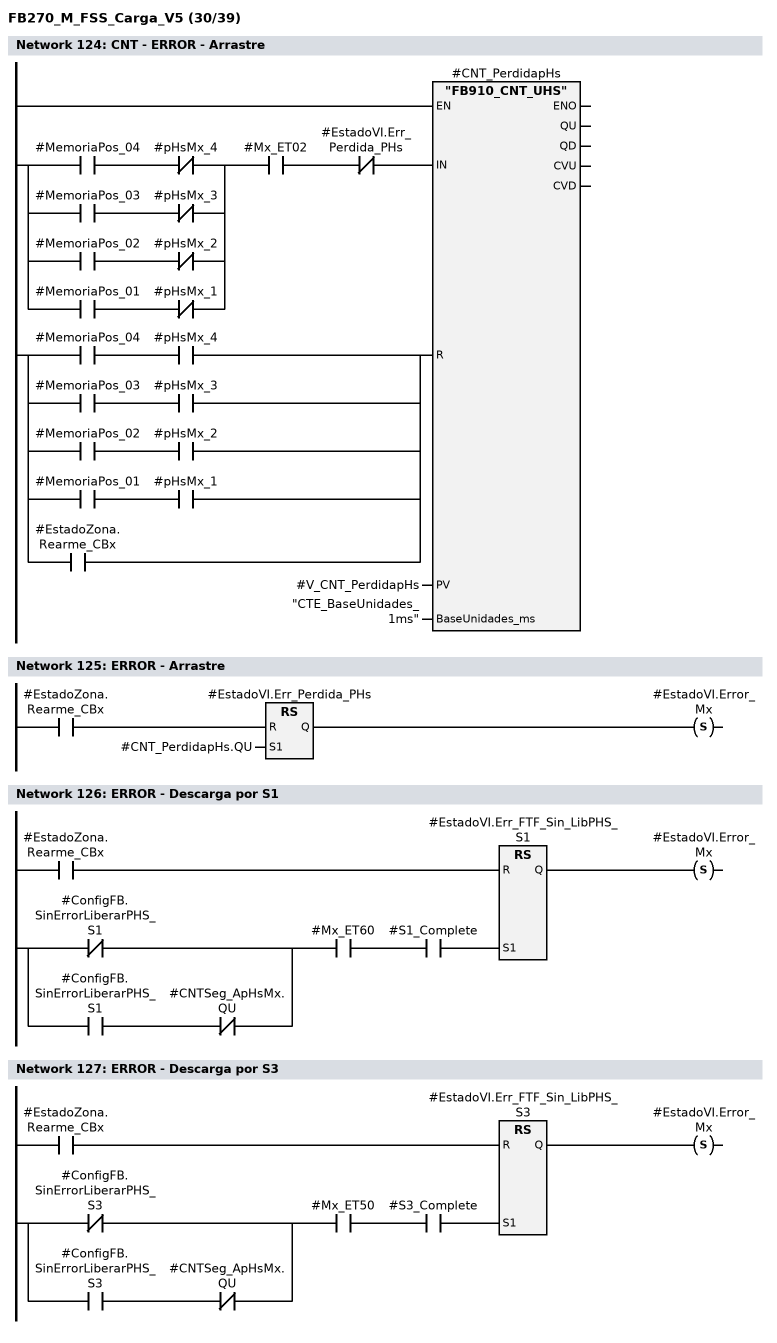
   RUNG wire#powerrail
      #CNT_PerdidapHs(IN := wire#w2, R := wire#w3, PV := #V_CNT_PerdidapHs, BaseUnidades_ms := "CTE_BaseUnidades_1ms", QU =>, QD =>, CVU =>, CVD =>)
   END_RUNG
   RUNG wire#powerrail
      Contact( #MemoriaPos_04 )
      I_Contact( #pHsMx_4 )
      wire#w1
      Contact( #Mx_ET02 )
      I_Contact( #EstadoVI.Err_Perdida_PHs )
   END_RUNG wire#w2
   RUNG wire#powerrail
      Contact( #MemoriaPos_03 )
      I_Contact( #pHsMx_3 )
   END_RUNG wire#w1
   RUNG wire#powerrail
      Contact( #MemoriaPos_02 )
      I_Contact( #pHsMx_2 )
   END_RUNG wire#w1
   RUNG wire#powerrail
      Contact( #MemoriaPos_01 )
      I_Contact( #pHsMx_1 )
   END_RUNG wire#w1
   RUNG wire#powerrail
      Contact( #MemoriaPos_04 )
      Contact( #pHsMx_4 )
   END_RUNG wire#w3
   RUNG wire#powerrail
      Contact( #MemoriaPos_03 )
      Contact( #pHsMx_3 )
   END_RUNG wire#w3
   RUNG wire#powerrail
      Contact( #MemoriaPos_02 )
      Contact( #pHsMx_2 )
   END_RUNG wire#w3
   RUNG wire#powerrail
      Contact( #MemoriaPos_01 )
      Contact( #pHsMx_1 )
   END_RUNG wire#w3
   RUNG wire#powerrail
      Contact( #EstadoZona.Rearme_CBx )
   END_RUNG wire#w3
   // the same network as SCL:
   #CNT_PerdidapHs(IN := ((#MemoriaPos_04 AND NOT #pHsMx_4) OR (#MemoriaPos_03 AND NOT #pHsMx_3) OR (#MemoriaPos_02 AND NOT #pHsMx_2) OR (#MemoriaPos_01 AND NOT #pHsMx_1)) AND #Mx_ET02 AND NOT #EstadoVI.Err_Perdida_PHs,   // "FB910_CNT_UHS"
                   R := (#MemoriaPos_04 AND #pHsMx_4) OR (#MemoriaPos_03 AND #pHsMx_3) OR (#MemoriaPos_02 AND #pHsMx_2) OR (#MemoriaPos_01 AND #pHsMx_1) OR #EstadoZona.Rearme_CBx,
                   PV := #V_CNT_PerdidapHs,
                   BaseUnidades_ms := "CTE_BaseUnidades_1ms");
END_REGION

REGION Network 125: ERROR - Arrastre
   RUNG wire#powerrail
      Contact( #EstadoZona.Rearme_CBx )
      S_RS(operand := #EstadoVI.Err_Perdida_PHs, s1 := #CNT_PerdidapHs.QU)
      S_Coil( #EstadoVI.Error_Mx )
   END_RUNG
   // the same network as SCL:
   IF #EstadoZona.Rearme_CBx THEN
       #EstadoVI.Err_Perdida_PHs := FALSE;   // RS flip-flop
   END_IF;
   IF #CNT_PerdidapHs.QU THEN #EstadoVI.Err_Perdida_PHs := TRUE; END_IF;
   IF #EstadoVI.Err_Perdida_PHs THEN #EstadoVI.Error_Mx := TRUE; END_IF;
END_REGION

REGION Network 126: ERROR - Descarga por S1
   RUNG wire#powerrail
      Contact( #EstadoZona.Rearme_CBx )
      S_RS(operand := #EstadoVI.Err_FTF_Sin_LibPHS_S1, s1 := wire#w2)
      S_Coil( #EstadoVI.Error_Mx )
   END_RUNG
   RUNG wire#powerrail
      I_Contact( #ConfigFB.SinErrorLiberarPHS_S1 )
      wire#w1
      Contact( #Mx_ET60 )
      Contact( #S1_Complete )
   END_RUNG wire#w2
   RUNG wire#powerrail
      Contact( #ConfigFB.SinErrorLiberarPHS_S1 )
      I_Contact( #CNTSeg_ApHsMx.QU )
   END_RUNG wire#w1
   // the same network as SCL:
   IF #EstadoZona.Rearme_CBx THEN
       #EstadoVI.Err_FTF_Sin_LibPHS_S1 := FALSE;   // RS flip-flop
   END_IF;
   IF (NOT #ConfigFB.SinErrorLiberarPHS_S1 OR (#ConfigFB.SinErrorLiberarPHS_S1 AND NOT #CNTSeg_ApHsMx.QU)) AND #Mx_ET60 AND #S1_Complete THEN
       #EstadoVI.Err_FTF_Sin_LibPHS_S1 := TRUE;
   END_IF;
   IF #EstadoVI.Err_FTF_Sin_LibPHS_S1 THEN #EstadoVI.Error_Mx := TRUE; END_IF;
END_REGION

REGION Network 127: ERROR - Descarga por S3
   RUNG wire#powerrail
      Contact( #EstadoZona.Rearme_CBx )
      S_RS(operand := #EstadoVI.Err_FTF_Sin_LibPHS_S3, s1 := wire#w2)
      S_Coil( #EstadoVI.Error_Mx )
   END_RUNG
   RUNG wire#powerrail
      I_Contact( #ConfigFB.SinErrorLiberarPHS_S3 )
      wire#w1
      Contact( #Mx_ET50 )
      Contact( #S3_Complete )
   END_RUNG wire#w2
   RUNG wire#powerrail
      Contact( #ConfigFB.SinErrorLiberarPHS_S3 )
      I_Contact( #CNTSeg_ApHsMx.QU )
   END_RUNG wire#w1
   // the same network as SCL:
   IF #EstadoZona.Rearme_CBx THEN
       #EstadoVI.Err_FTF_Sin_LibPHS_S3 := FALSE;   // RS flip-flop
   END_IF;
   IF (NOT #ConfigFB.SinErrorLiberarPHS_S3 OR (#ConfigFB.SinErrorLiberarPHS_S3 AND NOT #CNTSeg_ApHsMx.QU)) AND #Mx_ET50 AND #S3_Complete THEN
       #EstadoVI.Err_FTF_Sin_LibPHS_S3 := TRUE;
   END_IF;
   IF #EstadoVI.Err_FTF_Sin_LibPHS_S3 THEN #EstadoVI.Error_Mx := TRUE; END_IF;
END_REGION

REGION Network 128: TMP - ERROR - TimeOut Avance TRx >>> ENTRADA
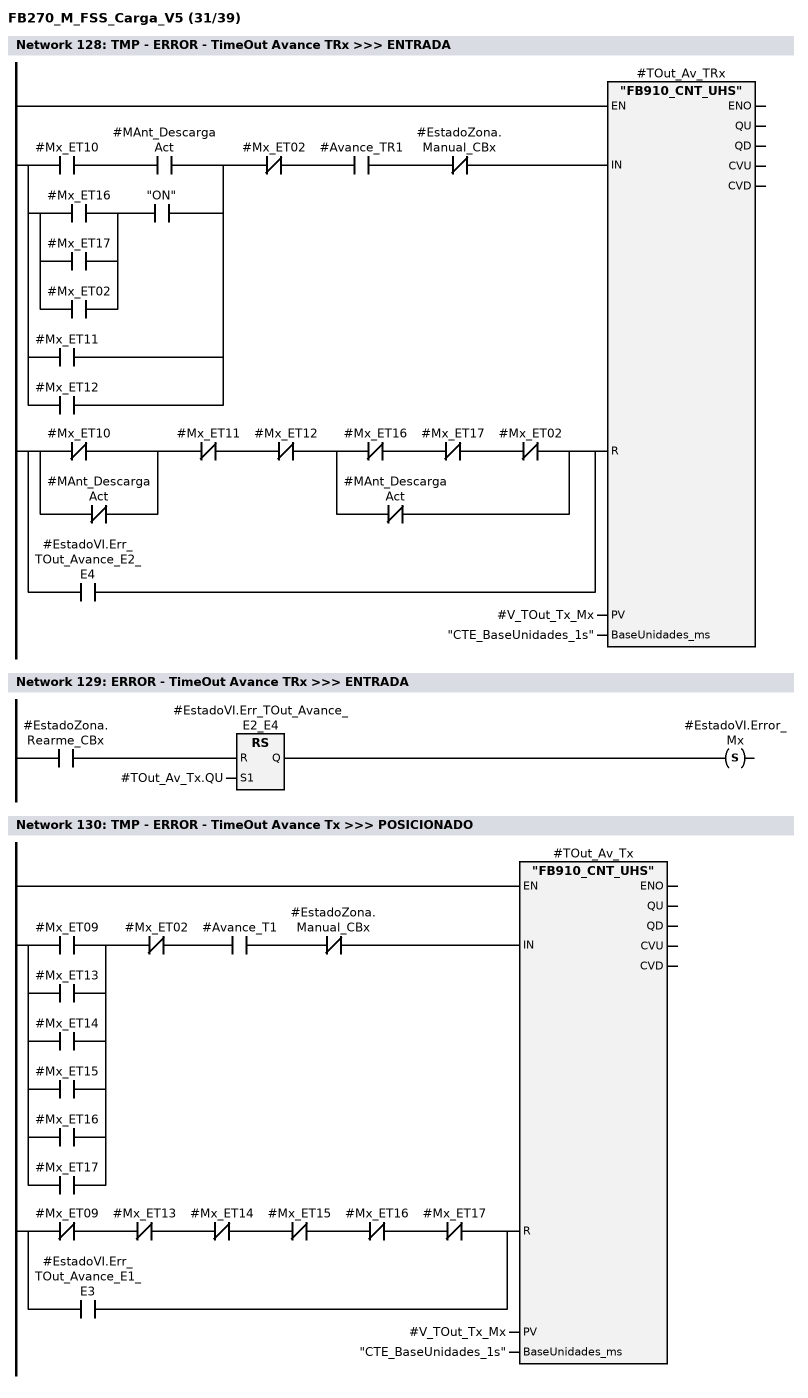
   RUNG wire#powerrail
      #TOut_Av_TRx(IN := wire#w3, R := wire#w6, PV := #V_TOut_Tx_Mx, BaseUnidades_ms := "CTE_BaseUnidades_1s", QU =>, QD =>, CVU =>, CVD =>)
   END_RUNG
   RUNG wire#powerrail
      Contact( #Mx_ET10 )
      Contact( #MAnt_DescargaAct )
      wire#w1
      I_Contact( #Mx_ET02 )
      Contact( #Avance_TR1 )
      I_Contact( #EstadoZona.Manual_CBx )
   END_RUNG wire#w3
   RUNG wire#powerrail
      Contact( #Mx_ET16 )
      wire#w2
      Contact( "ON" )
   END_RUNG wire#w1
   RUNG wire#powerrail
      Contact( #Mx_ET17 )
   END_RUNG wire#w2
   RUNG wire#powerrail
      Contact( #Mx_ET02 )
   END_RUNG wire#w2
   RUNG wire#powerrail
      Contact( #Mx_ET11 )
   END_RUNG wire#w1
   RUNG wire#powerrail
      Contact( #Mx_ET12 )
   END_RUNG wire#w1
   RUNG wire#powerrail
      I_Contact( #Mx_ET10 )
      wire#w4
      I_Contact( #Mx_ET11 )
      I_Contact( #Mx_ET12 )
      wire#w5
      I_Contact( #Mx_ET16 )
      I_Contact( #Mx_ET17 )
      I_Contact( #Mx_ET02 )
   END_RUNG wire#w6
   RUNG wire#powerrail
      I_Contact( #MAnt_DescargaAct )
   END_RUNG wire#w4
   RUNG wire#w5
      I_Contact( #MAnt_DescargaAct )
   END_RUNG wire#w6
   RUNG wire#powerrail
      Contact( #EstadoVI.Err_TOut_Avance_E2_E4 )
   END_RUNG wire#w6
   // the same network as SCL:
   #TOut_Av_TRx(IN := ((#Mx_ET10 AND #MAnt_DescargaAct) OR ((#Mx_ET16 OR #Mx_ET17 OR #Mx_ET02) AND "ON") OR #Mx_ET11 OR #Mx_ET12) AND NOT #Mx_ET02 AND #Avance_TR1 AND NOT #EstadoZona.Manual_CBx,   // "FB910_CNT_UHS"
                R := ((NOT #Mx_ET10 OR NOT #MAnt_DescargaAct) AND NOT #Mx_ET11 AND NOT #Mx_ET12 AND ((NOT #Mx_ET16 AND NOT #Mx_ET17 AND NOT #Mx_ET02) OR NOT #MAnt_DescargaAct)) OR #EstadoVI.Err_TOut_Avance_E2_E4,
                PV := #V_TOut_Tx_Mx,
                BaseUnidades_ms := "CTE_BaseUnidades_1s");
END_REGION

REGION Network 129: ERROR - TimeOut Avance TRx >>> ENTRADA
   RUNG wire#powerrail
      Contact( #EstadoZona.Rearme_CBx )
      S_RS(operand := #EstadoVI.Err_TOut_Avance_E2_E4, s1 := #TOut_Av_Tx.QU)
      S_Coil( #EstadoVI.Error_Mx )
   END_RUNG
   // the same network as SCL:
   IF #EstadoZona.Rearme_CBx THEN
       #EstadoVI.Err_TOut_Avance_E2_E4 := FALSE;   // RS flip-flop
   END_IF;
   IF #TOut_Av_Tx.QU THEN #EstadoVI.Err_TOut_Avance_E2_E4 := TRUE; END_IF;
   IF #EstadoVI.Err_TOut_Avance_E2_E4 THEN #EstadoVI.Error_Mx := TRUE; END_IF;
END_REGION

REGION Network 130: TMP - ERROR - TimeOut Avance Tx >>> POSICIONADO
   RUNG wire#powerrail
      #TOut_Av_Tx(IN := wire#w2, R := wire#w3, PV := #V_TOut_Tx_Mx, BaseUnidades_ms := "CTE_BaseUnidades_1s", QU =>, QD =>, CVU =>, CVD =>)
   END_RUNG
   RUNG wire#powerrail
      Contact( #Mx_ET09 )
      wire#w1
      I_Contact( #Mx_ET02 )
      Contact( #Avance_T1 )
      I_Contact( #EstadoZona.Manual_CBx )
   END_RUNG wire#w2
   RUNG wire#powerrail
      Contact( #Mx_ET13 )
   END_RUNG wire#w1
   RUNG wire#powerrail
      Contact( #Mx_ET14 )
   END_RUNG wire#w1
   RUNG wire#powerrail
      Contact( #Mx_ET15 )
   END_RUNG wire#w1
   RUNG wire#powerrail
      Contact( #Mx_ET16 )
   END_RUNG wire#w1
   RUNG wire#powerrail
      Contact( #Mx_ET17 )
   END_RUNG wire#w1
   RUNG wire#powerrail
      I_Contact( #Mx_ET09 )
      I_Contact( #Mx_ET13 )
      I_Contact( #Mx_ET14 )
      I_Contact( #Mx_ET15 )
      I_Contact( #Mx_ET16 )
      I_Contact( #Mx_ET17 )
   END_RUNG wire#w3
   RUNG wire#powerrail
      Contact( #EstadoVI.Err_TOut_Avance_E1_E3 )
   END_RUNG wire#w3
   // the same network as SCL:
   #TOut_Av_Tx(IN := (#Mx_ET09 OR #Mx_ET13 OR #Mx_ET14 OR #Mx_ET15 OR #Mx_ET16 OR #Mx_ET17) AND NOT #Mx_ET02 AND #Avance_T1 AND NOT #EstadoZona.Manual_CBx,   // "FB910_CNT_UHS"
               R := (NOT #Mx_ET09 AND NOT #Mx_ET13 AND NOT #Mx_ET14 AND NOT #Mx_ET15 AND NOT #Mx_ET16 AND NOT #Mx_ET17) OR #EstadoVI.Err_TOut_Avance_E1_E3,
               PV := #V_TOut_Tx_Mx,
               BaseUnidades_ms := "CTE_BaseUnidades_1s");
END_REGION

REGION Network 131: ERROR - TimeOut Avance Tx >>> POSICIONADO
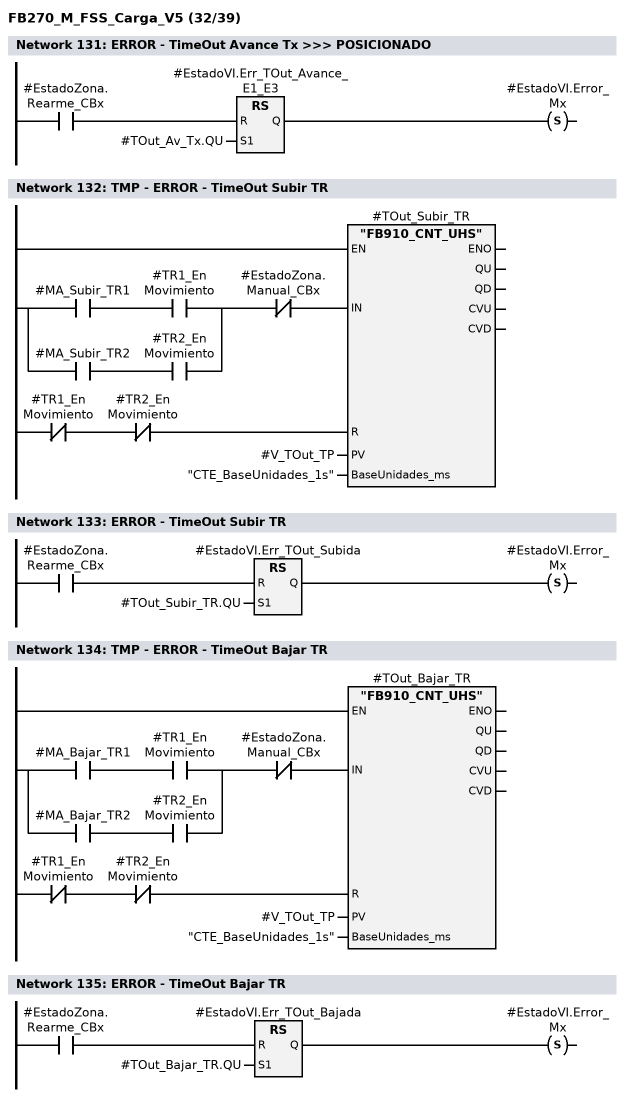
   RUNG wire#powerrail
      Contact( #EstadoZona.Rearme_CBx )
      S_RS(operand := #EstadoVI.Err_TOut_Avance_E1_E3, s1 := #TOut_Av_Tx.QU)
      S_Coil( #EstadoVI.Error_Mx )
   END_RUNG
   // the same network as SCL:
   IF #EstadoZona.Rearme_CBx THEN
       #EstadoVI.Err_TOut_Avance_E1_E3 := FALSE;   // RS flip-flop
   END_IF;
   IF #TOut_Av_Tx.QU THEN #EstadoVI.Err_TOut_Avance_E1_E3 := TRUE; END_IF;
   IF #EstadoVI.Err_TOut_Avance_E1_E3 THEN #EstadoVI.Error_Mx := TRUE; END_IF;
END_REGION

REGION Network 132: TMP - ERROR - TimeOut Subir TR
   RUNG wire#powerrail
      #TOut_Subir_TR(IN := wire#w2, R := wire#w3, PV := #V_TOut_TP, BaseUnidades_ms := "CTE_BaseUnidades_1s", QU =>, QD =>, CVU =>, CVD =>)
   END_RUNG
   RUNG wire#powerrail
      Contact( #MA_Subir_TR1 )
      Contact( #TR1_EnMovimiento )
      wire#w1
      I_Contact( #EstadoZona.Manual_CBx )
   END_RUNG wire#w2
   RUNG wire#powerrail
      Contact( #MA_Subir_TR2 )
      Contact( #TR2_EnMovimiento )
   END_RUNG wire#w1
   RUNG wire#powerrail
      I_Contact( #TR1_EnMovimiento )
      I_Contact( #TR2_EnMovimiento )
   END_RUNG wire#w3
   // the same network as SCL:
   #TOut_Subir_TR(IN := ((#MA_Subir_TR1 AND #TR1_EnMovimiento) OR (#MA_Subir_TR2 AND #TR2_EnMovimiento)) AND NOT #EstadoZona.Manual_CBx,   // "FB910_CNT_UHS"
                  R := NOT #TR1_EnMovimiento AND NOT #TR2_EnMovimiento,
                  PV := #V_TOut_TP,
                  BaseUnidades_ms := "CTE_BaseUnidades_1s");
END_REGION

REGION Network 133: ERROR - TimeOut Subir TR
   RUNG wire#powerrail
      Contact( #EstadoZona.Rearme_CBx )
      S_RS(operand := #EstadoVI.Err_TOut_Subida, s1 := #TOut_Subir_TR.QU)
      S_Coil( #EstadoVI.Error_Mx )
   END_RUNG
   // the same network as SCL:
   IF #EstadoZona.Rearme_CBx THEN
       #EstadoVI.Err_TOut_Subida := FALSE;   // RS flip-flop
   END_IF;
   IF #TOut_Subir_TR.QU THEN #EstadoVI.Err_TOut_Subida := TRUE; END_IF;
   IF #EstadoVI.Err_TOut_Subida THEN #EstadoVI.Error_Mx := TRUE; END_IF;
END_REGION

REGION Network 134: TMP - ERROR - TimeOut Bajar TR
   RUNG wire#powerrail
      #TOut_Bajar_TR(IN := wire#w2, R := wire#w3, PV := #V_TOut_TP, BaseUnidades_ms := "CTE_BaseUnidades_1s", QU =>, QD =>, CVU =>, CVD =>)
   END_RUNG
   RUNG wire#powerrail
      Contact( #MA_Bajar_TR1 )
      Contact( #TR1_EnMovimiento )
      wire#w1
      I_Contact( #EstadoZona.Manual_CBx )
   END_RUNG wire#w2
   RUNG wire#powerrail
      Contact( #MA_Bajar_TR2 )
      Contact( #TR2_EnMovimiento )
   END_RUNG wire#w1
   RUNG wire#powerrail
      I_Contact( #TR1_EnMovimiento )
      I_Contact( #TR2_EnMovimiento )
   END_RUNG wire#w3
   // the same network as SCL:
   #TOut_Bajar_TR(IN := ((#MA_Bajar_TR1 AND #TR1_EnMovimiento) OR (#MA_Bajar_TR2 AND #TR2_EnMovimiento)) AND NOT #EstadoZona.Manual_CBx,   // "FB910_CNT_UHS"
                  R := NOT #TR1_EnMovimiento AND NOT #TR2_EnMovimiento,
                  PV := #V_TOut_TP,
                  BaseUnidades_ms := "CTE_BaseUnidades_1s");
END_REGION

REGION Network 135: ERROR - TimeOut Bajar TR
   RUNG wire#powerrail
      Contact( #EstadoZona.Rearme_CBx )
      S_RS(operand := #EstadoVI.Err_TOut_Bajada, s1 := #TOut_Bajar_TR.QU)
      S_Coil( #EstadoVI.Error_Mx )
   END_RUNG
   // the same network as SCL:
   IF #EstadoZona.Rearme_CBx THEN
       #EstadoVI.Err_TOut_Bajada := FALSE;   // RS flip-flop
   END_IF;
   IF #TOut_Bajar_TR.QU THEN #EstadoVI.Err_TOut_Bajada := TRUE; END_IF;
   IF #EstadoVI.Err_TOut_Bajada THEN #EstadoVI.Error_Mx := TRUE; END_IF;
END_REGION

REGION Network 136: TMP - ERROR - TimeOut Subir TP E1E3
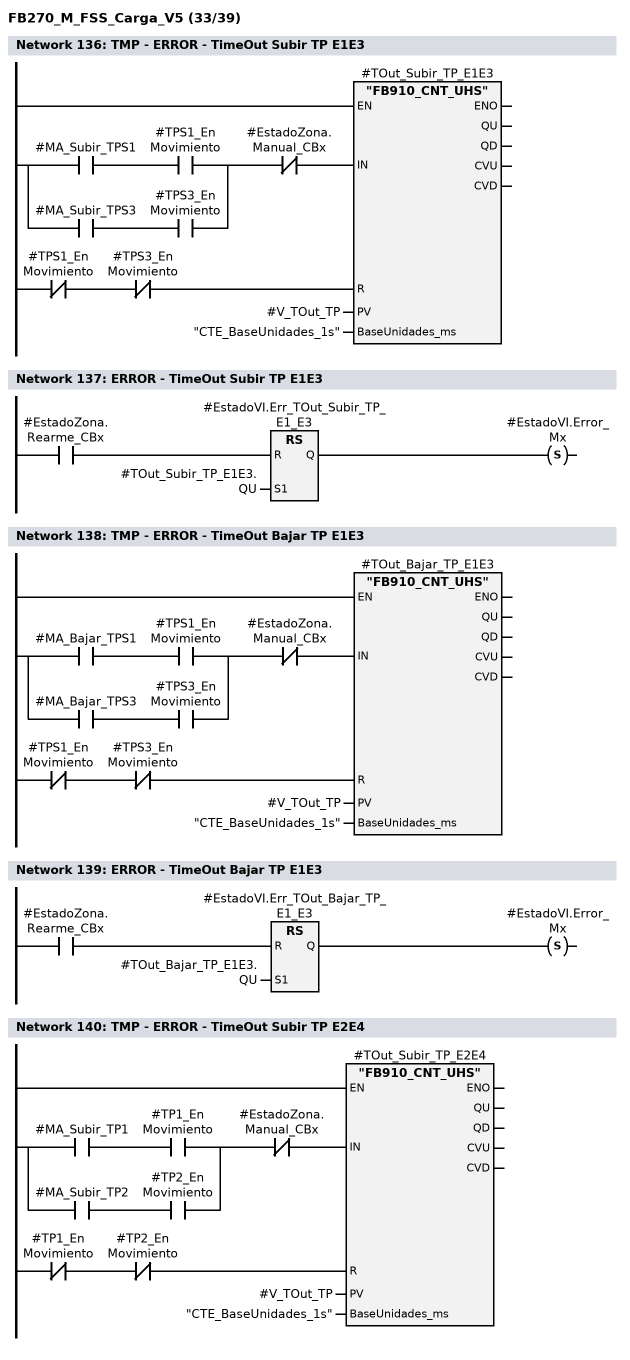
   RUNG wire#powerrail
      #TOut_Subir_TP_E1E3(IN := wire#w2, R := wire#w3, PV := #V_TOut_TP, BaseUnidades_ms := "CTE_BaseUnidades_1s", QU =>, QD =>, CVU =>, CVD =>)
   END_RUNG
   RUNG wire#powerrail
      Contact( #MA_Subir_TPS1 )
      Contact( #TPS1_EnMovimiento )
      wire#w1
      I_Contact( #EstadoZona.Manual_CBx )
   END_RUNG wire#w2
   RUNG wire#powerrail
      Contact( #MA_Subir_TPS3 )
      Contact( #TPS3_EnMovimiento )
   END_RUNG wire#w1
   RUNG wire#powerrail
      I_Contact( #TPS1_EnMovimiento )
      I_Contact( #TPS3_EnMovimiento )
   END_RUNG wire#w3
   // the same network as SCL:
   #TOut_Subir_TP_E1E3(IN := ((#MA_Subir_TPS1 AND #TPS1_EnMovimiento) OR (#MA_Subir_TPS3 AND #TPS3_EnMovimiento)) AND NOT #EstadoZona.Manual_CBx,   // "FB910_CNT_UHS"
                       R := NOT #TPS1_EnMovimiento AND NOT #TPS3_EnMovimiento,
                       PV := #V_TOut_TP,
                       BaseUnidades_ms := "CTE_BaseUnidades_1s");
END_REGION

REGION Network 137: ERROR - TimeOut Subir TP E1E3
   RUNG wire#powerrail
      Contact( #EstadoZona.Rearme_CBx )
      S_RS(operand := #EstadoVI.Err_TOut_Subir_TP_E1_E3, s1 := #TOut_Subir_TP_E1E3.QU)
      S_Coil( #EstadoVI.Error_Mx )
   END_RUNG
   // the same network as SCL:
   IF #EstadoZona.Rearme_CBx THEN
       #EstadoVI.Err_TOut_Subir_TP_E1_E3 := FALSE;   // RS flip-flop
   END_IF;
   IF #TOut_Subir_TP_E1E3.QU THEN #EstadoVI.Err_TOut_Subir_TP_E1_E3 := TRUE; END_IF;
   IF #EstadoVI.Err_TOut_Subir_TP_E1_E3 THEN #EstadoVI.Error_Mx := TRUE; END_IF;
END_REGION

REGION Network 138: TMP - ERROR - TimeOut Bajar TP E1E3
   RUNG wire#powerrail
      #TOut_Bajar_TP_E1E3(IN := wire#w2, R := wire#w3, PV := #V_TOut_TP, BaseUnidades_ms := "CTE_BaseUnidades_1s", QU =>, QD =>, CVU =>, CVD =>)
   END_RUNG
   RUNG wire#powerrail
      Contact( #MA_Bajar_TPS1 )
      Contact( #TPS1_EnMovimiento )
      wire#w1
      I_Contact( #EstadoZona.Manual_CBx )
   END_RUNG wire#w2
   RUNG wire#powerrail
      Contact( #MA_Bajar_TPS3 )
      Contact( #TPS3_EnMovimiento )
   END_RUNG wire#w1
   RUNG wire#powerrail
      I_Contact( #TPS1_EnMovimiento )
      I_Contact( #TPS3_EnMovimiento )
   END_RUNG wire#w3
   // the same network as SCL:
   #TOut_Bajar_TP_E1E3(IN := ((#MA_Bajar_TPS1 AND #TPS1_EnMovimiento) OR (#MA_Bajar_TPS3 AND #TPS3_EnMovimiento)) AND NOT #EstadoZona.Manual_CBx,   // "FB910_CNT_UHS"
                       R := NOT #TPS1_EnMovimiento AND NOT #TPS3_EnMovimiento,
                       PV := #V_TOut_TP,
                       BaseUnidades_ms := "CTE_BaseUnidades_1s");
END_REGION

REGION Network 139: ERROR - TimeOut Bajar TP E1E3
   RUNG wire#powerrail
      Contact( #EstadoZona.Rearme_CBx )
      S_RS(operand := #EstadoVI.Err_TOut_Bajar_TP_E1_E3, s1 := #TOut_Bajar_TP_E1E3.QU)
      S_Coil( #EstadoVI.Error_Mx )
   END_RUNG
   // the same network as SCL:
   IF #EstadoZona.Rearme_CBx THEN
       #EstadoVI.Err_TOut_Bajar_TP_E1_E3 := FALSE;   // RS flip-flop
   END_IF;
   IF #TOut_Bajar_TP_E1E3.QU THEN #EstadoVI.Err_TOut_Bajar_TP_E1_E3 := TRUE; END_IF;
   IF #EstadoVI.Err_TOut_Bajar_TP_E1_E3 THEN #EstadoVI.Error_Mx := TRUE; END_IF;
END_REGION

REGION Network 140: TMP - ERROR - TimeOut Subir TP E2E4
   RUNG wire#powerrail
      #TOut_Subir_TP_E2E4(IN := wire#w2, R := wire#w3, PV := #V_TOut_TP, BaseUnidades_ms := "CTE_BaseUnidades_1s", QU =>, QD =>, CVU =>, CVD =>)
   END_RUNG
   RUNG wire#powerrail
      Contact( #MA_Subir_TP1 )
      Contact( #TP1_EnMovimiento )
      wire#w1
      I_Contact( #EstadoZona.Manual_CBx )
   END_RUNG wire#w2
   RUNG wire#powerrail
      Contact( #MA_Subir_TP2 )
      Contact( #TP2_EnMovimiento )
   END_RUNG wire#w1
   RUNG wire#powerrail
      I_Contact( #TP1_EnMovimiento )
      I_Contact( #TP2_EnMovimiento )
   END_RUNG wire#w3
   // the same network as SCL:
   #TOut_Subir_TP_E2E4(IN := ((#MA_Subir_TP1 AND #TP1_EnMovimiento) OR (#MA_Subir_TP2 AND #TP2_EnMovimiento)) AND NOT #EstadoZona.Manual_CBx,   // "FB910_CNT_UHS"
                       R := NOT #TP1_EnMovimiento AND NOT #TP2_EnMovimiento,
                       PV := #V_TOut_TP,
                       BaseUnidades_ms := "CTE_BaseUnidades_1s");
END_REGION

REGION Network 141: ERROR - TimeOut Subir TP E2E4
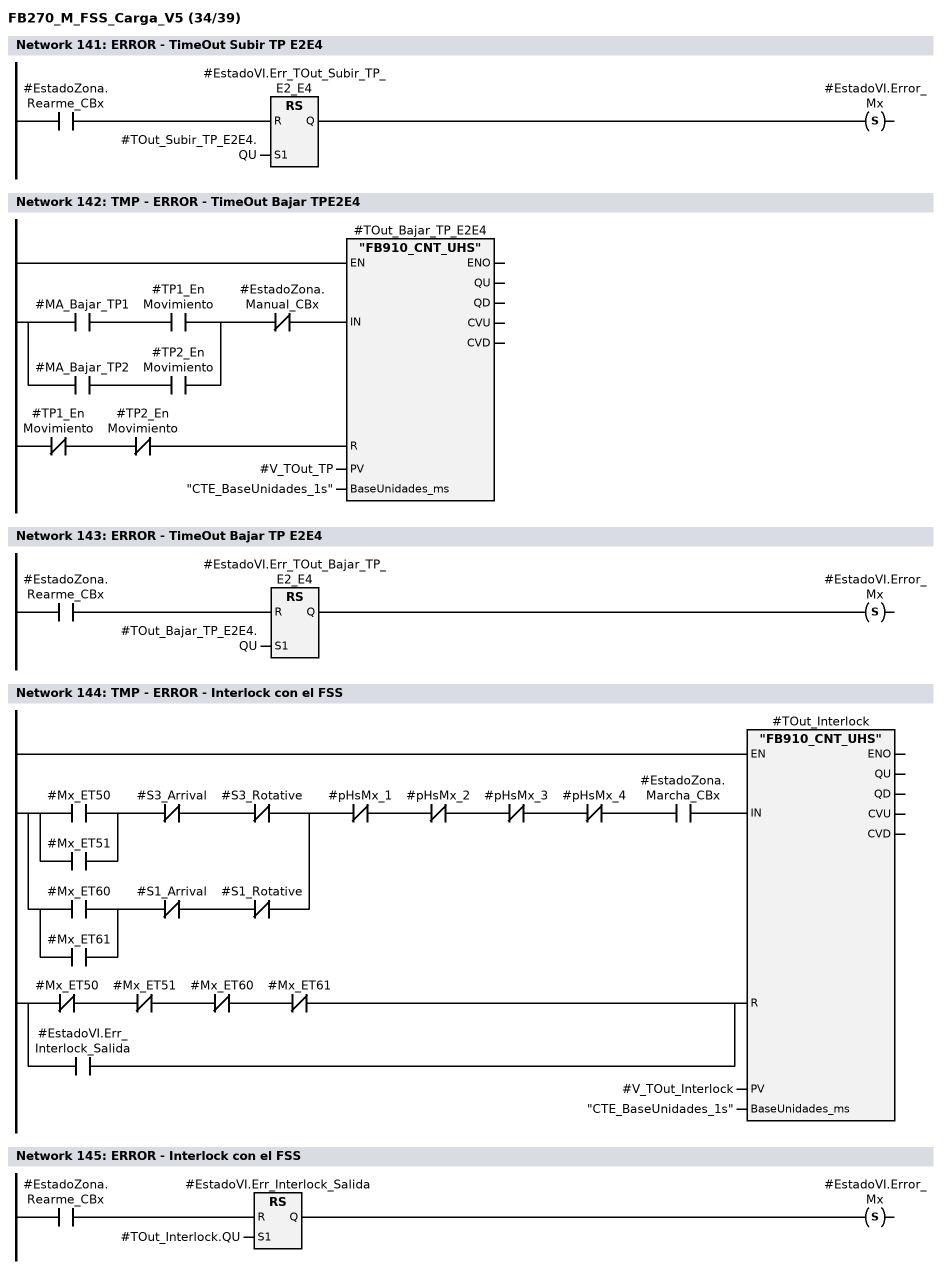
   RUNG wire#powerrail
      Contact( #EstadoZona.Rearme_CBx )
      S_RS(operand := #EstadoVI.Err_TOut_Subir_TP_E2_E4, s1 := #TOut_Subir_TP_E2E4.QU)
      S_Coil( #EstadoVI.Error_Mx )
   END_RUNG
   // the same network as SCL:
   IF #EstadoZona.Rearme_CBx THEN
       #EstadoVI.Err_TOut_Subir_TP_E2_E4 := FALSE;   // RS flip-flop
   END_IF;
   IF #TOut_Subir_TP_E2E4.QU THEN #EstadoVI.Err_TOut_Subir_TP_E2_E4 := TRUE; END_IF;
   IF #EstadoVI.Err_TOut_Subir_TP_E2_E4 THEN #EstadoVI.Error_Mx := TRUE; END_IF;
END_REGION

REGION Network 142: TMP - ERROR - TimeOut Bajar TPE2E4
   RUNG wire#powerrail
      #TOut_Bajar_TP_E2E4(IN := wire#w2, R := wire#w3, PV := #V_TOut_TP, BaseUnidades_ms := "CTE_BaseUnidades_1s", QU =>, QD =>, CVU =>, CVD =>)
   END_RUNG
   RUNG wire#powerrail
      Contact( #MA_Bajar_TP1 )
      Contact( #TP1_EnMovimiento )
      wire#w1
      I_Contact( #EstadoZona.Manual_CBx )
   END_RUNG wire#w2
   RUNG wire#powerrail
      Contact( #MA_Bajar_TP2 )
      Contact( #TP2_EnMovimiento )
   END_RUNG wire#w1
   RUNG wire#powerrail
      I_Contact( #TP1_EnMovimiento )
      I_Contact( #TP2_EnMovimiento )
   END_RUNG wire#w3
   // the same network as SCL:
   #TOut_Bajar_TP_E2E4(IN := ((#MA_Bajar_TP1 AND #TP1_EnMovimiento) OR (#MA_Bajar_TP2 AND #TP2_EnMovimiento)) AND NOT #EstadoZona.Manual_CBx,   // "FB910_CNT_UHS"
                       R := NOT #TP1_EnMovimiento AND NOT #TP2_EnMovimiento,
                       PV := #V_TOut_TP,
                       BaseUnidades_ms := "CTE_BaseUnidades_1s");
END_REGION

REGION Network 143: ERROR - TimeOut Bajar TP E2E4
   RUNG wire#powerrail
      Contact( #EstadoZona.Rearme_CBx )
      S_RS(operand := #EstadoVI.Err_TOut_Bajar_TP_E2_E4, s1 := #TOut_Bajar_TP_E2E4.QU)
      S_Coil( #EstadoVI.Error_Mx )
   END_RUNG
   // the same network as SCL:
   IF #EstadoZona.Rearme_CBx THEN
       #EstadoVI.Err_TOut_Bajar_TP_E2_E4 := FALSE;   // RS flip-flop
   END_IF;
   IF #TOut_Bajar_TP_E2E4.QU THEN #EstadoVI.Err_TOut_Bajar_TP_E2_E4 := TRUE; END_IF;
   IF #EstadoVI.Err_TOut_Bajar_TP_E2_E4 THEN #EstadoVI.Error_Mx := TRUE; END_IF;
END_REGION

REGION Network 144: TMP - ERROR - Interlock con el FSS
   RUNG wire#powerrail
      #TOut_Interlock(IN := wire#w4, R := wire#w5, PV := #V_TOut_Interlock, BaseUnidades_ms := "CTE_BaseUnidades_1s", QU =>, QD =>, CVU =>, CVD =>)
   END_RUNG
   RUNG wire#powerrail
      Contact( #Mx_ET50 )
      wire#w1
      I_Contact( #S3_Arrival )
      I_Contact( #S3_Rotative )
      wire#w2
      I_Contact( #pHsMx_1 )
      I_Contact( #pHsMx_2 )
      I_Contact( #pHsMx_3 )
      I_Contact( #pHsMx_4 )
      Contact( #EstadoZona.Marcha_CBx )
   END_RUNG wire#w4
   RUNG wire#powerrail
      Contact( #Mx_ET51 )
   END_RUNG wire#w1
   RUNG wire#powerrail
      Contact( #Mx_ET60 )
      wire#w3
      I_Contact( #S1_Arrival )
      I_Contact( #S1_Rotative )
   END_RUNG wire#w2
   RUNG wire#powerrail
      Contact( #Mx_ET61 )
   END_RUNG wire#w3
   RUNG wire#powerrail
      I_Contact( #Mx_ET50 )
      I_Contact( #Mx_ET51 )
      I_Contact( #Mx_ET60 )
      I_Contact( #Mx_ET61 )
   END_RUNG wire#w5
   RUNG wire#powerrail
      Contact( #EstadoVI.Err_Interlock_Salida )
   END_RUNG wire#w5
   // the same network as SCL:
   #TOut_Interlock(IN := (((#Mx_ET50 OR #Mx_ET51) AND NOT #S3_Arrival AND NOT #S3_Rotative) OR ((#Mx_ET60 OR #Mx_ET61) AND NOT #S1_Arrival AND NOT #S1_Rotative)) AND NOT #pHsMx_1 AND NOT #pHsMx_2 AND NOT #pHsMx_3 AND NOT #pHsMx_4 AND #EstadoZona.Marcha_CBx,   // "FB910_CNT_UHS"
                   R := (NOT #Mx_ET50 AND NOT #Mx_ET51 AND NOT #Mx_ET60 AND NOT #Mx_ET61) OR #EstadoVI.Err_Interlock_Salida,
                   PV := #V_TOut_Interlock,
                   BaseUnidades_ms := "CTE_BaseUnidades_1s");
END_REGION

REGION Network 145: ERROR - Interlock con el FSS
   RUNG wire#powerrail
      Contact( #EstadoZona.Rearme_CBx )
      S_RS(operand := #EstadoVI.Err_Interlock_Salida, s1 := #TOut_Interlock.QU)
      S_Coil( #EstadoVI.Error_Mx )
   END_RUNG
   // the same network as SCL:
   IF #EstadoZona.Rearme_CBx THEN
       #EstadoVI.Err_Interlock_Salida := FALSE;   // RS flip-flop
   END_IF;
   IF #TOut_Interlock.QU THEN #EstadoVI.Err_Interlock_Salida := TRUE; END_IF;
   IF #EstadoVI.Err_Interlock_Salida THEN #EstadoVI.Error_Mx := TRUE; END_IF;
END_REGION

REGION Network 146: ESTADOS DE LA MESA
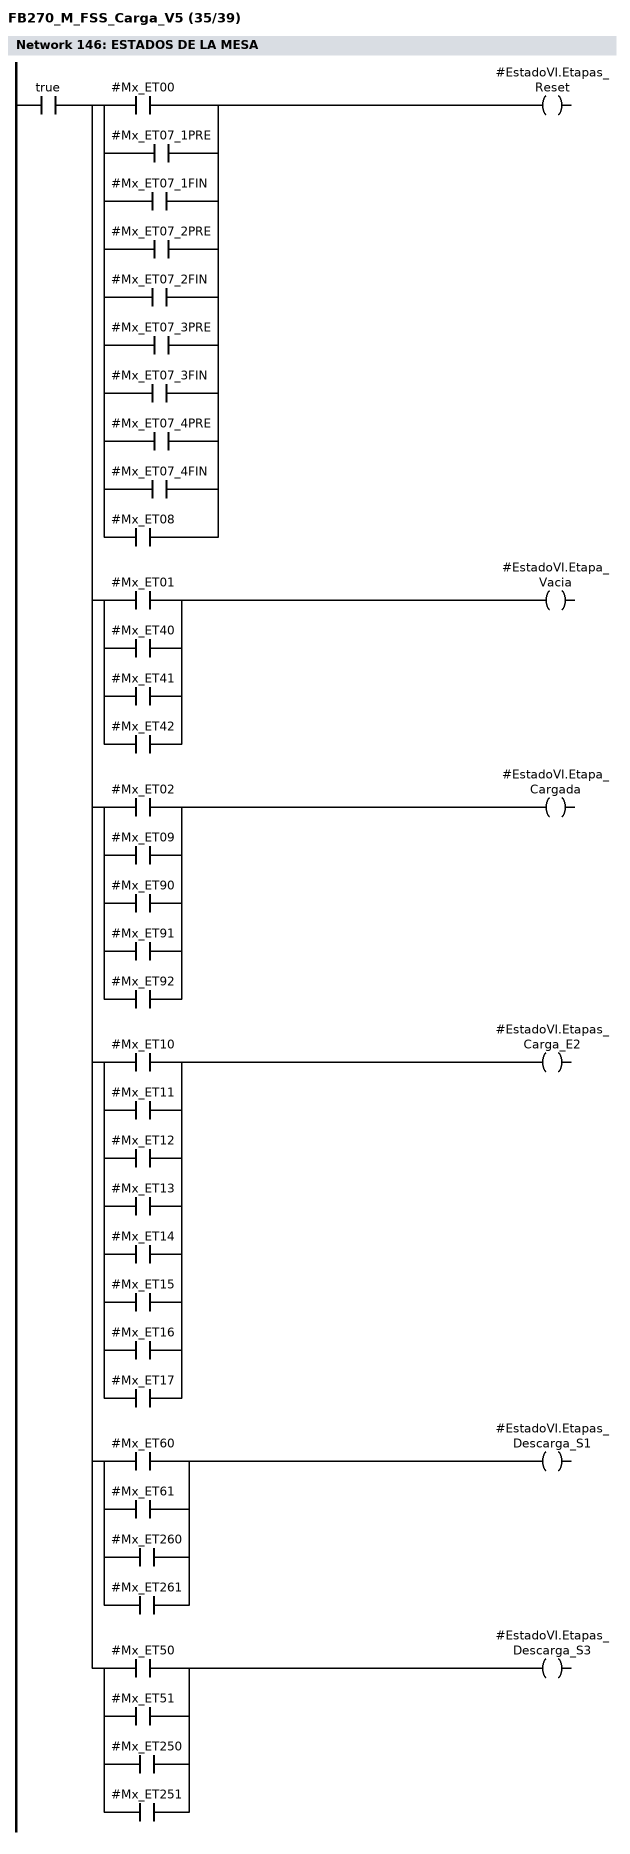
   RUNG wire#powerrail
      Contact( true )
      wire#w1
      Contact( #Mx_ET00 )
      wire#w2
      Coil( #EstadoVI.Etapas_Reset )
   END_RUNG
   RUNG wire#w1
      Contact( #Mx_ET07_1PRE )
   END_RUNG wire#w2
   RUNG wire#w1
      Contact( #Mx_ET07_1FIN )
   END_RUNG wire#w2
   RUNG wire#w1
      Contact( #Mx_ET07_2PRE )
   END_RUNG wire#w2
   RUNG wire#w1
      Contact( #Mx_ET07_2FIN )
   END_RUNG wire#w2
   RUNG wire#w1
      Contact( #Mx_ET07_3PRE )
   END_RUNG wire#w2
   RUNG wire#w1
      Contact( #Mx_ET07_3FIN )
   END_RUNG wire#w2
   RUNG wire#w1
      Contact( #Mx_ET07_4PRE )
   END_RUNG wire#w2
   RUNG wire#w1
      Contact( #Mx_ET07_4FIN )
   END_RUNG wire#w2
   RUNG wire#w1
      Contact( #Mx_ET08 )
   END_RUNG wire#w2
   RUNG wire#w1
      Contact( #Mx_ET01 )
      wire#w3
      Coil( #EstadoVI.Etapa_Vacia )
   END_RUNG
   RUNG wire#w1
      Contact( #Mx_ET40 )
   END_RUNG wire#w3
   RUNG wire#w1
      Contact( #Mx_ET41 )
   END_RUNG wire#w3
   RUNG wire#w1
      Contact( #Mx_ET42 )
   END_RUNG wire#w3
   RUNG wire#w1
      Contact( #Mx_ET02 )
      wire#w4
      Coil( #EstadoVI.Etapa_Cargada )
   END_RUNG
   RUNG wire#w1
      Contact( #Mx_ET09 )
   END_RUNG wire#w4
   RUNG wire#w1
      Contact( #Mx_ET90 )
   END_RUNG wire#w4
   RUNG wire#w1
      Contact( #Mx_ET91 )
   END_RUNG wire#w4
   RUNG wire#w1
      Contact( #Mx_ET92 )
   END_RUNG wire#w4
   RUNG wire#w1
      Contact( #Mx_ET10 )
      wire#w5
      Coil( #EstadoVI.Etapas_Carga_E2 )
   END_RUNG
   RUNG wire#w1
      Contact( #Mx_ET11 )
   END_RUNG wire#w5
   RUNG wire#w1
      Contact( #Mx_ET12 )
   END_RUNG wire#w5
   RUNG wire#w1
      Contact( #Mx_ET13 )
   END_RUNG wire#w5
   RUNG wire#w1
      Contact( #Mx_ET14 )
   END_RUNG wire#w5
   RUNG wire#w1
      Contact( #Mx_ET15 )
   END_RUNG wire#w5
   RUNG wire#w1
      Contact( #Mx_ET16 )
   END_RUNG wire#w5
   RUNG wire#w1
      Contact( #Mx_ET17 )
   END_RUNG wire#w5
   RUNG wire#w1
      Contact( #Mx_ET60 )
      wire#w6
      Coil( #EstadoVI.Etapas_Descarga_S1 )
   END_RUNG
   RUNG wire#w1
      Contact( #Mx_ET61 )
   END_RUNG wire#w6
   RUNG wire#w1
      Contact( #Mx_ET260 )
   END_RUNG wire#w6
   RUNG wire#w1
      Contact( #Mx_ET261 )
   END_RUNG wire#w6
   RUNG wire#w1
      Contact( #Mx_ET50 )
      wire#w7
      Coil( #EstadoVI.Etapas_Descarga_S3 )
   END_RUNG
   RUNG wire#w1
      Contact( #Mx_ET51 )
   END_RUNG wire#w7
   RUNG wire#w1
      Contact( #Mx_ET250 )
   END_RUNG wire#w7
   RUNG wire#w1
      Contact( #Mx_ET251 )
   END_RUNG wire#w7
   // the same network as SCL:
   #EstadoVI.Etapas_Reset := true AND (#Mx_ET00 OR #Mx_ET07_1PRE OR #Mx_ET07_1FIN OR #Mx_ET07_2PRE OR #Mx_ET07_2FIN OR #Mx_ET07_3PRE OR #Mx_ET07_3FIN OR #Mx_ET07_4PRE OR #Mx_ET07_4FIN OR #Mx_ET08);
   #EstadoVI.Etapa_Vacia := true AND (#Mx_ET01 OR #Mx_ET40 OR #Mx_ET41 OR #Mx_ET42);
   #EstadoVI.Etapa_Cargada := true AND (#Mx_ET02 OR #Mx_ET09 OR #Mx_ET90 OR #Mx_ET91 OR #Mx_ET92);
   #EstadoVI.Etapas_Carga_E2 := true AND (#Mx_ET10 OR #Mx_ET11 OR #Mx_ET12 OR #Mx_ET13 OR #Mx_ET14 OR #Mx_ET15 OR #Mx_ET16 OR #Mx_ET17);
   #EstadoVI.Etapas_Descarga_S1 := true AND (#Mx_ET60 OR #Mx_ET61 OR #Mx_ET260 OR #Mx_ET261);
   #EstadoVI.Etapas_Descarga_S3 := true AND (#Mx_ET50 OR #Mx_ET51 OR #Mx_ET250 OR #Mx_ET251);
END_REGION

REGION Network 147: ENTRADAS DE LA MESA
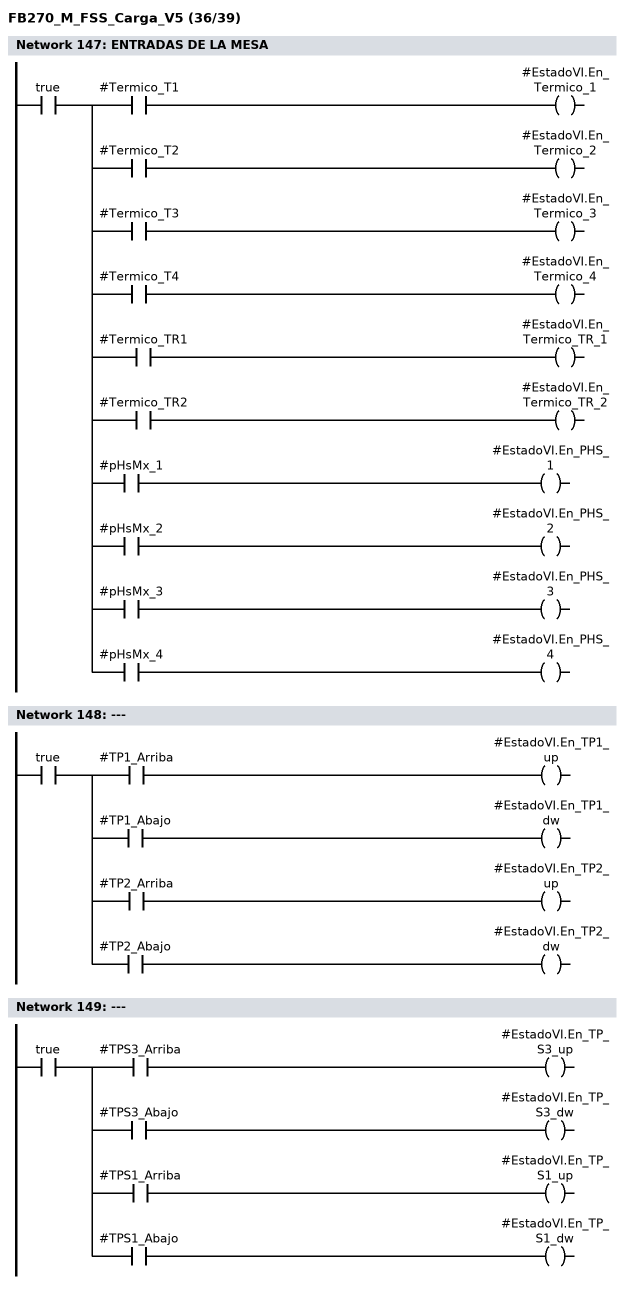
   RUNG wire#powerrail
      Contact( true )
      wire#w1
      Contact( #Termico_T1 )
      Coil( #EstadoVI.En_Termico_1 )
   END_RUNG
   RUNG wire#w1
      Contact( #Termico_T2 )
      Coil( #EstadoVI.En_Termico_2 )
   END_RUNG
   RUNG wire#w1
      Contact( #Termico_T3 )
      Coil( #EstadoVI.En_Termico_3 )
   END_RUNG
   RUNG wire#w1
      Contact( #Termico_T4 )
      Coil( #EstadoVI.En_Termico_4 )
   END_RUNG
   RUNG wire#w1
      Contact( #Termico_TR1 )
      Coil( #EstadoVI.En_Termico_TR_1 )
   END_RUNG
   RUNG wire#w1
      Contact( #Termico_TR2 )
      Coil( #EstadoVI.En_Termico_TR_2 )
   END_RUNG
   RUNG wire#w1
      Contact( #pHsMx_1 )
      Coil( #EstadoVI.En_PHS_1 )
   END_RUNG
   RUNG wire#w1
      Contact( #pHsMx_2 )
      Coil( #EstadoVI.En_PHS_2 )
   END_RUNG
   RUNG wire#w1
      Contact( #pHsMx_3 )
      Coil( #EstadoVI.En_PHS_3 )
   END_RUNG
   RUNG wire#w1
      Contact( #pHsMx_4 )
      Coil( #EstadoVI.En_PHS_4 )
   END_RUNG
   // the same network as SCL:
   #EstadoVI.En_Termico_1 := true AND #Termico_T1;
   #EstadoVI.En_Termico_2 := true AND #Termico_T2;
   #EstadoVI.En_Termico_3 := true AND #Termico_T3;
   #EstadoVI.En_Termico_4 := true AND #Termico_T4;
   #EstadoVI.En_Termico_TR_1 := true AND #Termico_TR1;
   #EstadoVI.En_Termico_TR_2 := true AND #Termico_TR2;
   #EstadoVI.En_PHS_1 := true AND #pHsMx_1;
   #EstadoVI.En_PHS_2 := true AND #pHsMx_2;
   #EstadoVI.En_PHS_3 := true AND #pHsMx_3;
   #EstadoVI.En_PHS_4 := true AND #pHsMx_4;
END_REGION

REGION Network 148: ---
   RUNG wire#powerrail
      Contact( true )
      wire#w1
      Contact( #TP1_Arriba )
      Coil( #EstadoVI.En_TP1_up )
   END_RUNG
   RUNG wire#w1
      Contact( #TP1_Abajo )
      Coil( #EstadoVI.En_TP1_dw )
   END_RUNG
   RUNG wire#w1
      Contact( #TP2_Arriba )
      Coil( #EstadoVI.En_TP2_up )
   END_RUNG
   RUNG wire#w1
      Contact( #TP2_Abajo )
      Coil( #EstadoVI.En_TP2_dw )
   END_RUNG
   // the same network as SCL:
   #EstadoVI.En_TP1_up := true AND #TP1_Arriba;
   #EstadoVI.En_TP1_dw := true AND #TP1_Abajo;
   #EstadoVI.En_TP2_up := true AND #TP2_Arriba;
   #EstadoVI.En_TP2_dw := true AND #TP2_Abajo;
END_REGION

REGION Network 149: ---
   RUNG wire#powerrail
      Contact( true )
      wire#w1
      Contact( #TPS3_Arriba )
      Coil( #EstadoVI.En_TP_S3_up )
   END_RUNG
   RUNG wire#w1
      Contact( #TPS3_Abajo )
      Coil( #EstadoVI.En_TP_S3_dw )
   END_RUNG
   RUNG wire#w1
      Contact( #TPS1_Arriba )
      Coil( #EstadoVI.En_TP_S1_up )
   END_RUNG
   RUNG wire#w1
      Contact( #TPS1_Abajo )
      Coil( #EstadoVI.En_TP_S1_dw )
   END_RUNG
   // the same network as SCL:
   #EstadoVI.En_TP_S3_up := true AND #TPS3_Arriba;
   #EstadoVI.En_TP_S3_dw := true AND #TPS3_Abajo;
   #EstadoVI.En_TP_S1_up := true AND #TPS1_Arriba;
   #EstadoVI.En_TP_S1_dw := true AND #TPS1_Abajo;
END_REGION

REGION Network 150: ---
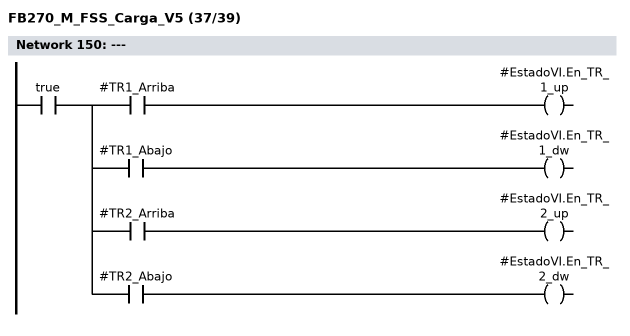
   RUNG wire#powerrail
      Contact( true )
      wire#w1
      Contact( #TR1_Arriba )
      Coil( #EstadoVI.En_TR_1_up )
   END_RUNG
   RUNG wire#w1
      Contact( #TR1_Abajo )
      Coil( #EstadoVI.En_TR_1_dw )
   END_RUNG
   RUNG wire#w1
      Contact( #TR2_Arriba )
      Coil( #EstadoVI.En_TR_2_up )
   END_RUNG
   RUNG wire#w1
      Contact( #TR2_Abajo )
      Coil( #EstadoVI.En_TR_2_dw )
   END_RUNG
   // the same network as SCL:
   #EstadoVI.En_TR_1_up := true AND #TR1_Arriba;
   #EstadoVI.En_TR_1_dw := true AND #TR1_Abajo;
   #EstadoVI.En_TR_2_up := true AND #TR2_Arriba;
   #EstadoVI.En_TR_2_dw := true AND #TR2_Abajo;
END_REGION

REGION Network 151: SALIDAS DE LA MESA
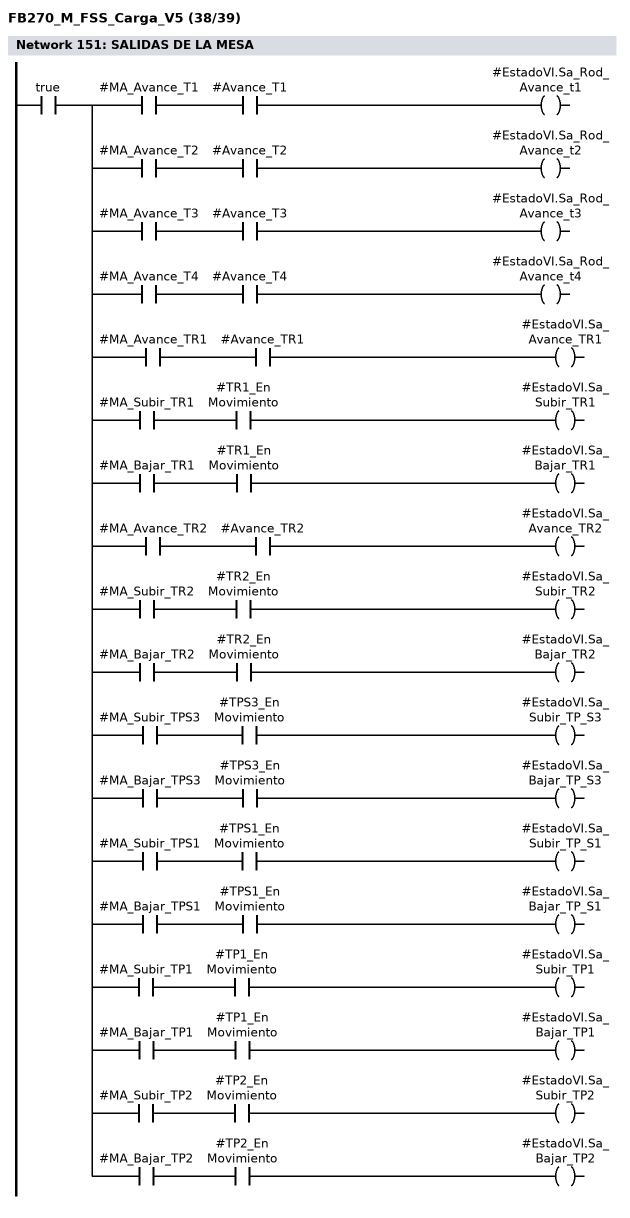
   RUNG wire#powerrail
      Contact( true )
      wire#w1
      Contact( #MA_Avance_T1 )
      Contact( #Avance_T1 )
      Coil( #EstadoVI.Sa_Rod_Avance_t1 )
   END_RUNG
   RUNG wire#w1
      Contact( #MA_Avance_T2 )
      Contact( #Avance_T2 )
      Coil( #EstadoVI.Sa_Rod_Avance_t2 )
   END_RUNG
   RUNG wire#w1
      Contact( #MA_Avance_T3 )
      Contact( #Avance_T3 )
      Coil( #EstadoVI.Sa_Rod_Avance_t3 )
   END_RUNG
   RUNG wire#w1
      Contact( #MA_Avance_T4 )
      Contact( #Avance_T4 )
      Coil( #EstadoVI.Sa_Rod_Avance_t4 )
   END_RUNG
   RUNG wire#w1
      Contact( #MA_Avance_TR1 )
      Contact( #Avance_TR1 )
      Coil( #EstadoVI.Sa_Avance_TR1 )
   END_RUNG
   RUNG wire#w1
      Contact( #MA_Subir_TR1 )
      Contact( #TR1_EnMovimiento )
      Coil( #EstadoVI.Sa_Subir_TR1 )
   END_RUNG
   RUNG wire#w1
      Contact( #MA_Bajar_TR1 )
      Contact( #TR1_EnMovimiento )
      Coil( #EstadoVI.Sa_Bajar_TR1 )
   END_RUNG
   RUNG wire#w1
      Contact( #MA_Avance_TR2 )
      Contact( #Avance_TR2 )
      Coil( #EstadoVI.Sa_Avance_TR2 )
   END_RUNG
   RUNG wire#w1
      Contact( #MA_Subir_TR2 )
      Contact( #TR2_EnMovimiento )
      Coil( #EstadoVI.Sa_Subir_TR2 )
   END_RUNG
   RUNG wire#w1
      Contact( #MA_Bajar_TR2 )
      Contact( #TR2_EnMovimiento )
      Coil( #EstadoVI.Sa_Bajar_TR2 )
   END_RUNG
   RUNG wire#w1
      Contact( #MA_Subir_TPS3 )
      Contact( #TPS3_EnMovimiento )
      Coil( #EstadoVI.Sa_Subir_TP_S3 )
   END_RUNG
   RUNG wire#w1
      Contact( #MA_Bajar_TPS3 )
      Contact( #TPS3_EnMovimiento )
      Coil( #EstadoVI.Sa_Bajar_TP_S3 )
   END_RUNG
   RUNG wire#w1
      Contact( #MA_Subir_TPS1 )
      Contact( #TPS1_EnMovimiento )
      Coil( #EstadoVI.Sa_Subir_TP_S1 )
   END_RUNG
   RUNG wire#w1
      Contact( #MA_Bajar_TPS1 )
      Contact( #TPS1_EnMovimiento )
      Coil( #EstadoVI.Sa_Bajar_TP_S1 )
   END_RUNG
   RUNG wire#w1
      Contact( #MA_Subir_TP1 )
      Contact( #TP1_EnMovimiento )
      Coil( #EstadoVI.Sa_Subir_TP1 )
   END_RUNG
   RUNG wire#w1
      Contact( #MA_Bajar_TP1 )
      Contact( #TP1_EnMovimiento )
      Coil( #EstadoVI.Sa_Bajar_TP1 )
   END_RUNG
   RUNG wire#w1
      Contact( #MA_Subir_TP2 )
      Contact( #TP2_EnMovimiento )
      Coil( #EstadoVI.Sa_Subir_TP2 )
   END_RUNG
   RUNG wire#w1
      Contact( #MA_Bajar_TP2 )
      Contact( #TP2_EnMovimiento )
      Coil( #EstadoVI.Sa_Bajar_TP2 )
   END_RUNG
   // the same network as SCL:
   #EstadoVI.Sa_Rod_Avance_t1 := true AND #MA_Avance_T1 AND #Avance_T1;
   #EstadoVI.Sa_Rod_Avance_t2 := true AND #MA_Avance_T2 AND #Avance_T2;
   #EstadoVI.Sa_Rod_Avance_t3 := true AND #MA_Avance_T3 AND #Avance_T3;
   #EstadoVI.Sa_Rod_Avance_t4 := true AND #MA_Avance_T4 AND #Avance_T4;
   #EstadoVI.Sa_Avance_TR1 := true AND #MA_Avance_TR1 AND #Avance_TR1;
   #EstadoVI.Sa_Subir_TR1 := true AND #MA_Subir_TR1 AND #TR1_EnMovimiento;
   #EstadoVI.Sa_Bajar_TR1 := true AND #MA_Bajar_TR1 AND #TR1_EnMovimiento;
   #EstadoVI.Sa_Avance_TR2 := true AND #MA_Avance_TR2 AND #Avance_TR2;
   #EstadoVI.Sa_Subir_TR2 := true AND #MA_Subir_TR2 AND #TR2_EnMovimiento;
   #EstadoVI.Sa_Bajar_TR2 := true AND #MA_Bajar_TR2 AND #TR2_EnMovimiento;
   #EstadoVI.Sa_Subir_TP_S3 := true AND #MA_Subir_TPS3 AND #TPS3_EnMovimiento;
   #EstadoVI.Sa_Bajar_TP_S3 := true AND #MA_Bajar_TPS3 AND #TPS3_EnMovimiento;
   #EstadoVI.Sa_Subir_TP_S1 := true AND #MA_Subir_TPS1 AND #TPS1_EnMovimiento;
   #EstadoVI.Sa_Bajar_TP_S1 := true AND #MA_Bajar_TPS1 AND #TPS1_EnMovimiento;
   #EstadoVI.Sa_Subir_TP1 := true AND #MA_Subir_TP1 AND #TP1_EnMovimiento;
   #EstadoVI.Sa_Bajar_TP1 := true AND #MA_Bajar_TP1 AND #TP1_EnMovimiento;
   #EstadoVI.Sa_Subir_TP2 := true AND #MA_Subir_TP2 AND #TP2_EnMovimiento;
   #EstadoVI.Sa_Bajar_TP2 := true AND #MA_Bajar_TP2 AND #TP2_EnMovimiento;
END_REGION

REGION Network 152: INTERLOCK PARA HMI
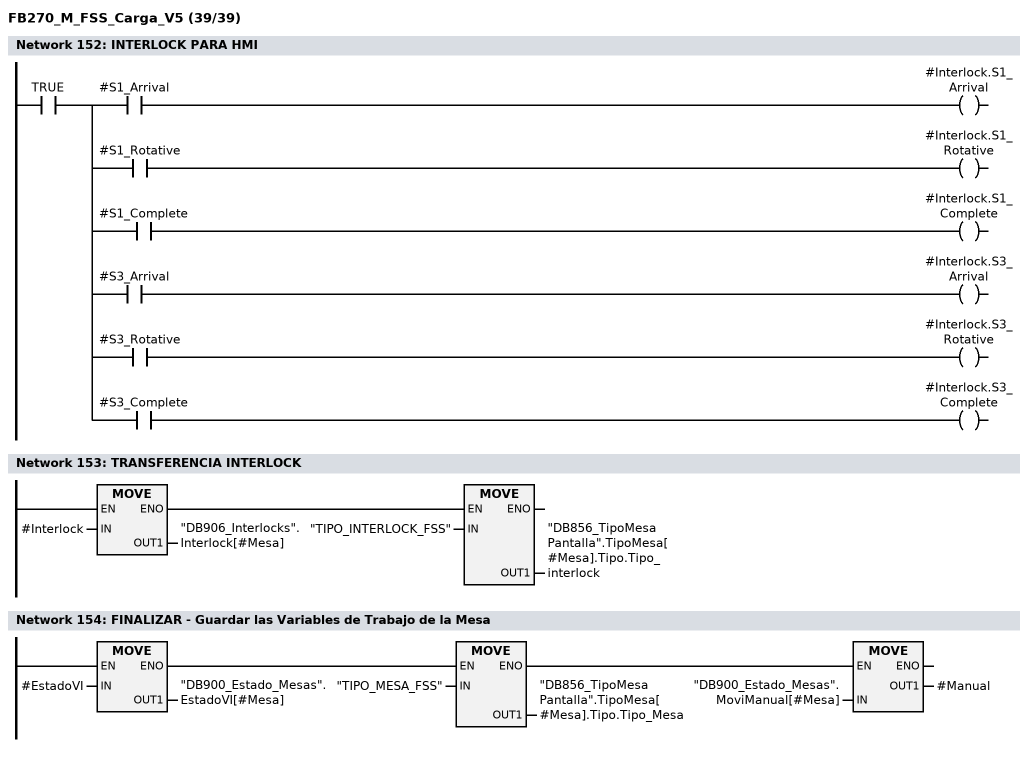
   RUNG wire#powerrail
      Contact( TRUE )
      wire#w1
      Contact( #S1_Arrival )
      Coil( #Interlock.S1_Arrival )
   END_RUNG
   RUNG wire#w1
      Contact( #S1_Rotative )
      Coil( #Interlock.S1_Rotative )
   END_RUNG
   RUNG wire#w1
      Contact( #S1_Complete )
      Coil( #Interlock.S1_Complete )
   END_RUNG
   RUNG wire#w1
      Contact( #S3_Arrival )
      Coil( #Interlock.S3_Arrival )
   END_RUNG
   RUNG wire#w1
      Contact( #S3_Rotative )
      Coil( #Interlock.S3_Rotative )
   END_RUNG
   RUNG wire#w1
      Contact( #S3_Complete )
      Coil( #Interlock.S3_Complete )
   END_RUNG
   // the same network as SCL:
   #Interlock.S1_Arrival := TRUE AND #S1_Arrival;
   #Interlock.S1_Rotative := TRUE AND #S1_Rotative;
   #Interlock.S1_Complete := TRUE AND #S1_Complete;
   #Interlock.S3_Arrival := TRUE AND #S3_Arrival;
   #Interlock.S3_Rotative := TRUE AND #S3_Rotative;
   #Interlock.S3_Complete := TRUE AND #S3_Complete;
END_REGION

REGION Network 153: TRANSFERENCIA INTERLOCK
   RUNG wire#powerrail
      Move(in := #Interlock, out1 => "DB906_Interlocks".Interlock[#Mesa])
      Move(in := "TIPO_INTERLOCK_FSS", out1 => "DB856_TipoMesaPantalla".TipoMesa[#Mesa].Tipo.Tipo_interlock)
   END_RUNG
   // the same network as SCL:
   "DB906_Interlocks".Interlock[#Mesa] := #Interlock;
   "DB856_TipoMesaPantalla".TipoMesa[#Mesa].Tipo.Tipo_interlock := "TIPO_INTERLOCK_FSS";
END_REGION

REGION Network 154: FINALIZAR - Guardar las Variables de Trabajo de la Mesa
   RUNG wire#powerrail
      Move(in := #EstadoVI, out1 => "DB900_Estado_Mesas".EstadoVI[#Mesa])
      Move(in := "TIPO_MESA_FSS", out1 => "DB856_TipoMesaPantalla".TipoMesa[#Mesa].Tipo.Tipo_Mesa)
      Move(in := "DB900_Estado_Mesas".MoviManual[#Mesa], out1 => #Manual)
   END_RUNG
   // the same network as SCL:
   "DB900_Estado_Mesas".EstadoVI[#Mesa] := #EstadoVI;
   "DB856_TipoMesaPantalla".TipoMesa[#Mesa].Tipo.Tipo_Mesa := "TIPO_MESA_FSS";
   #Manual := "DB900_Estado_Mesas".MoviManual[#Mesa];
END_REGION
END_FUNCTION_BLOCK
